// TwinCAT 3 PLC project Untitled1
// Title: RobustSolution
// Company: BATW
// Author: BATW
// ProjectVersion: 1.0.0.1
// ProgramVersion: 3.1.4026.24
// libraries:
//   Tc2_MC2, * (Beckhoff Automation GmbH)
//   Tc2_Standard, * (Beckhoff Automation GmbH)
//   Tc2_System, * (Beckhoff Automation GmbH)
//   Tc2_Utilities, * (Beckhoff Automation GmbH)
//   Tc3_JsonXml, * (Beckhoff Automation GmbH)
//   TcUnit, * (www.tcunit.org)
// project tree:
//   Configuration/DUTs/ E_AlarmOperator.TcDUT (not stored), E_ConfigDataType.TcDUT, E_ConfigValueError.TcDUT (not stored), E_LinkPhase.TcDUT (not stored), E_ModuleType.TcDUT, T_ModuleTypeName.TcDUT (not stored), E_VariableAccess.TcDUT, ST_ConfigRawValue.TcDUT (not stored), ST_ReferenceBindingFileConfig.TcDUT, ST_ConfigAlarmInfo.TcDUT (not stored), ST_ConfigVariableInfo.TcDUT (not stored), ST_RuntimeAlarmBinding.TcDUT (not stored), ST_RuntimeVariableBinding.TcDUT (not stored), ST_LinkVariableNode.TcDUT, ST_MappingFileConfig.TcDUT, ST_ModuleFileConfig.TcDUT, ST_ModuleRuntimeConfig.TcDUT, ST_SystemFileConfig.TcDUT, ST_VariableLink.TcDUT (not stored)
//   Configuration/POUs/ F_AlarmConditionMet.TcPOU, F_ConfigDataTypeSize.TcPOU, F_ConfigDataTypeToDescriptor.TcPOU (not stored), F_ConfigValueErrorMessage.TcPOU, FB_ConfigValueSnapshotReader.TcPOU, FB_ModuleTypeRegistry.TcPOU, FB_ReferenceManager.TcPOU, FB_ModuleReferenceBindingContext.TcPOU, FB_LinkVariableManager.TcPOU, FB_ModuleConfigurationManager.TcPOU, FB_ApplicationConfigRoot.TcPOU
//   Configuration/Interfaces/ I_AdsSymbolProvider.TcIO, I_ModuleReferenceBindings.TcIO, I_ModuleConfigurationAdapter.TcIO, I_VariableNodeReader.TcIO
//   DUTs/Contracts/Alarm/ E_Severity.TcDUT (not stored), ST_ExtAlarm.TcDUT (not stored)
//   DUTs/Contracts/Descriptor/ E_DescriptorType.TcDUT (not stored), ST_ExtDescriptor.TcDUT
//   DUTs/Contracts/System/ ST_SystemContext.TcDUT
//   DUTs/Infrastructure/EL Modules/ ST_EL1889Ex.TcDUT (not stored), ST_EL2809Ex.TcDUT (not stored), ST_EL3602Ex.TcDUT (not stored)
//   DUTs/Infrastructure/ ST_ReserveForGetSymbolNameByAddrress.TcDUT (not stored)
//   DUTs/Module/Alarm/ E_AlarmAckCommand.TcDUT (not stored), E_AlarmAckError.TcDUT (not stored), ST_AlarmAckRequest.TcDUT (not stored), ST_AlarmLifecycleState.TcDUT (not stored), ST_ModuleAlarmStatus.TcDUT (not stored)
//   DUTs/Module/Contract/ ST_ModuleCtrl.TcDUT (not stored), ST_ModuleDataStatus.TcDUT (not stored), ST_ModuleStatus.TcDUT (not stored), ST_ModuleVariableStatus.TcDUT, ST_Module_CtrlStatus_Base.TcDUT (not stored)
//   DUTs/Module/ServiceCoordination/ E_CompositeOwnershipState.TcDUT, E_ServiceCallSubmitResult.TcDUT, E_ServiceInternalCommandState.TcDUT (not stored), E_ServiceRegistrationError.TcDUT, ST_ServiceExecutionSnapshot.TcDUT, ST_ServiceRegistrationEntry.TcDUT
//   DUTs/Service/Composite/ E_CompositeServiceErrorCode.TcDUT
//   DUTs/Service/Contracts/ E_ServiceCompletionBehavior.TcDUT (not stored), ST_ServiceContext.TcDUT (not stored), ST_ServiceCtrl.TcDUT (not stored), ST_ServiceDataStatus.TcDUT, ST_ServiceExecuteSubStateRecord.TcDUT (not stored), ST_ServiceExecuteSubStateStatus.TcDUT, ST_ServiceStatus.TcDUT (not stored)
//   DUTs/Wafer Transfer/ E_OperationState.TcDUT (not stored), E_ReceiveState.TcDUT, E_TransferCapability.TcDUT, E_WaferHandlingType.TcDUT, ST_TransferHandshakeSignal.TcDUT, ST_MaterialContext.TcDUT, ST_MaterialInfo.TcDUT, ST_WaferTransferCtrl.TcDUT, ST_WaferTransferParam.TcDUT, ST_WaferTransferStatus.TcDUT, ST_WaferTransferResponse.TcDUT, ST_WaferTransferRequest.TcDUT
//   GVLs/ Param_Config.TcGVL
//   / PlcTask.TcTTO
//   POUs/00_BaseUnit/Base/ FB_BaseUnit.TcPOU (not stored), T_ResourceOwnerId.TcDUT (not stored)
//   POUs/00_BaseUnit/ FB_Axis_BaseUnit.TcPOU
//   POUs/00_BaseUnit/Interfaces/ I_Axis_BaseUnit.TcIO, I_BaseUnit.TcIO, I_ResourceLock.TcIO
//   POUs/10_Module/ FB_ModuleAlarmManager.TcPOU, FB_ModuleBase.TcPOU, FB_ServiceCoordinator.TcPOU, FB_ServiceCaller.TcPOU
//   POUs/20_Service/ FB_CompositeServiceBase.TcPOU (not stored), FB_ServiceBase.TcPOU (not stored)
//   POUs/ FB_UtcClock.TcPOU (not stored)
//   POUs/30_PackML_Base/DUTs/ E_PackMLCommand.TcDUT (not stored), E_PackMLErrorID.TcDUT (not stored), E_PackMLHookResult.TcDUT (not stored), E_PackMLMode.TcDUT (not stored), E_PackMLState.TcDUT (not stored), ST_PML_Base_In.TcDUT (not stored), ST_PML_Base_Out.TcDUT (not stored), T_PackMLMode.TcDUT
//   POUs/30_PackML_Base/ FB_PackMLBase.TcPOU, FB_PackMLModeSet.TcPOU (not stored)
//   POUs/30_PackML_Base/Utilities/ F_PackMLCommandToString.TcPOU (not stored), F_PackMLErrorIDToString.TcPOU (not stored), F_PackMLModeToString.TcPOU (not stored), F_PackMLStateToString.TcPOU (not stored)
// real-time tasks:
//   TASK PlcTask: cycle T#10ms, priority 20, ADS port 350

CONFIGURATION Untitled1
    RESOURCE PLC ON TwinCAT3
        TASK PlcTask(INTERVAL := T#10ms, PRIORITY := 20);
    END_RESOURCE
END_CONFIGURATION

// ---- Configuration/DUTs/E_ConfigDataType.TcDUT
{attribute 'qualified_only'}
{attribute 'strict'}
{attribute 'to_string'}
TYPE E_ConfigDataType :
(
	Unknown := 0,
	Boolean,
	Integer32,
	UnsignedInteger32,
	Float32,
	Float64,
	String80
);
END_TYPE

// ---- Configuration/DUTs/E_ModuleType.TcDUT
{attribute 'qualified_only'}
{attribute 'strict'}
{attribute 'to_string'}
TYPE E_ModuleType :
(
	Unknown := 0,
	// Chamber1 Module. The member name is the public config value.
	Chamber1 := 1
);
END_TYPE

// ---- Configuration/DUTs/E_VariableAccess.TcDUT
{attribute 'qualified_only'}
{attribute 'strict'}
TYPE E_VariableAccess :
(
	ReadOnly := 1,
	WriteOnly,
	ReadWrite
);
END_TYPE

// ---- Configuration/DUTs/ST_ReferenceBindingFileConfig.TcDUT
TYPE ST_ReferenceBindingFileConfig :
STRUCT
	Name : STRING(80);
	Source : STRING(255);
END_STRUCT
END_TYPE

// ---- Configuration/DUTs/ST_LinkVariableNode.TcDUT
TYPE ST_LinkVariableNode :
STRUCT
	Name : STRING(255);
	Address : PVOID;
	Size : UDINT;
	DataType : E_ConfigDataType;
	Access : E_VariableAccess;
END_STRUCT
END_TYPE

// ---- Configuration/DUTs/ST_MappingFileConfig.TcDUT
TYPE ST_MappingFileConfig :
STRUCT
	Source : STRING(255);
	Target : STRING(255);
	SourceDataType : E_ConfigDataType;
	TargetDataType : E_ConfigDataType;
	HasTransform : BOOL;
	Scale : LREAL;
	Offset : LREAL;
END_STRUCT
END_TYPE

// ---- Configuration/DUTs/ST_ModuleFileConfig.TcDUT
TYPE ST_ModuleFileConfig :
STRUCT
	Enabled : BOOL;
	Slot : UINT;
	Id : UDINT;
	ModuleType : T_ModuleTypeName;
	InputMappingCount : UINT;
	InputMappings : ARRAY[1..Param_Config.MaxModuleMappings] OF ST_MappingFileConfig;
	OutputMappingCount : UINT;
	OutputMappings : ARRAY[1..Param_Config.MaxModuleMappings] OF ST_MappingFileConfig;
	ReferenceCount : UINT;
	References : ARRAY[1..Param_Config.MaxModuleReferences] OF ST_ReferenceBindingFileConfig;
	VariableCount : UINT;
	VariableList : ARRAY[1..Param_Config.MaxModuleVariable] OF ST_ConfigVariableInfo;
	AlarmCount : UINT;
	AlarmList : ARRAY[1..Param_Config.MaxConfiguredAlarmsPerModule] OF ST_ConfigAlarmInfo;
END_STRUCT
END_TYPE

// ---- Configuration/DUTs/ST_ModuleRuntimeConfig.TcDUT
TYPE ST_ModuleRuntimeConfig :
STRUCT
	Enabled : BOOL;
	Valid : BOOL;
	ModuleId : UDINT;
	ModuleType : T_ModuleTypeName;
	Revision : UDINT;
	VariableCount : UINT;
	VariableBindings : ARRAY[1..Param_Config.MaxModuleVariable] OF ST_RuntimeVariableBinding;
	AlarmCount : UINT;
	AlarmBindings : ARRAY[1..Param_Config.MaxConfiguredAlarmsPerModule] OF ST_RuntimeAlarmBinding;
END_STRUCT
END_TYPE

// ---- Configuration/DUTs/ST_SystemFileConfig.TcDUT
TYPE ST_SystemFileConfig :
STRUCT
	SchemaVersion : UDINT;
	ModuleCount : UINT;
	Modules : ARRAY[1..Param_Config.MaxTotalConfiguredModules] OF ST_ModuleFileConfig;
END_STRUCT
END_TYPE

// ---- DUTs/Contracts/Descriptor/ST_ExtDescriptor.TcDUT
TYPE ST_ExtDescriptor :
STRUCT
	Id : UDINT;
	Name : STRING(30);
	DataType : E_DescriptorType;
	Unit : STRING(10);
	Value : STRING(80);
END_STRUCT
END_TYPE

// ---- DUTs/Contracts/System/ST_SystemContext.TcDUT
TYPE ST_SystemContext :
STRUCT
	// UTC timestamp formatted as YYYYMMDDHHMMSSUUU.
	UtcDateTime : STRING(20);
	// Maximum time that a Module may observe an unchanged HeartbeatIndex.
	ModuleHeartbeatTimeout : TIME;
END_STRUCT
END_TYPE

// ---- DUTs/Module/Contract/ST_ModuleVariableStatus.TcDUT
TYPE ST_ModuleVariableStatus :
STRUCT
	PublishedCount : UINT;
	Overflow : BOOL;
	DuplicateId : UDINT;
END_STRUCT
END_TYPE

// ---- DUTs/Module/ServiceCoordination/E_CompositeOwnershipState.TcDUT
{attribute 'qualified_only'}
{attribute 'strict'}
{attribute 'to_string'}
TYPE E_CompositeOwnershipState :
(
	None := 0,
	Pending := 1,
	Owned := 2,
	RejectedConflict := 3,
	RejectedDependencyNotIdle := 4,
	RejectedUnsupportedCompletionBehavior := 5,
	Cancelled := 6
) UDINT;
END_TYPE

// ---- DUTs/Module/ServiceCoordination/E_ServiceCallSubmitResult.TcDUT
{attribute 'qualified_only'}
{attribute 'strict'}
{attribute 'to_string'}
TYPE E_ServiceCallSubmitResult :
(
	Queued := 0,
	CallerNotConfigured := 1,
	CoordinatorNotReady := 2,
	UnknownService := 3,
	DependencyNotDeclared := 4,
	NotOwner := 5,
	Busy := 6,
	InvalidCommand := 7,
	ParameterSizeMismatch := 8,
	ParameterTypeResolutionFailed := 9,
	ParameterTypeMismatch := 10
) UDINT;
END_TYPE

// ---- DUTs/Module/ServiceCoordination/E_ServiceRegistrationError.TcDUT
{attribute 'qualified_only'}
{attribute 'strict'}
{attribute 'to_string'}
TYPE E_ServiceRegistrationError :
(
	None := 0,
	RegistrationAlreadyStarted := 1,
	RegistryAlreadySealed := 2,
	EmptyRegistry := 3,
	CapacityExceeded := 4,
	InvalidServiceId := 5,
	DuplicateServiceId := 6,
	InvalidStorage := 7,
	ParameterSizeMismatch := 8,
	ParameterTypeMismatch := 9,
	ParameterTypeResolutionFailed := 10,
	InvalidCompositeService := 11,
	DuplicateCompositeDefinition := 12,
	EmptyCompositeDependencyList := 13,
	CompositeDependencyCapacityExceeded := 14,
	InvalidCompositeDependencyId := 15,
	UnknownCompositeDependency := 16,
	SelfDependency := 17,
	DuplicateCompositeDependency := 18,
	CompositeDependencyNotAllowed := 19,
	NestedCompositeNotSupported := 20
) UDINT;
END_TYPE

// ---- DUTs/Module/ServiceCoordination/ST_ServiceExecutionSnapshot.TcDUT
TYPE ST_ServiceExecutionSnapshot :
STRUCT
	Valid : BOOL;
	ServiceId : UDINT;
	ResponseId : UDINT;
	PackMLOut : ST_PML_Base_Out;
	ExecuteSubState : UDINT;
	CompletionBehavior : E_ServiceCompletionBehavior;
END_STRUCT
END_TYPE

// ---- DUTs/Module/ServiceCoordination/ST_ServiceRegistrationEntry.TcDUT
TYPE ST_ServiceRegistrationEntry :
STRUCT
	InUse : BOOL;
	ServiceId : UDINT;

	UpperCtrlAddress : PVOID;
	EffectiveCtrlAddress : PVOID;

	UpperParamAddress : PVOID;
	EffectiveParamAddress : PVOID;
	ParameterSize : UDINT;
	ParameterTypeName : STRING(255);

	StatusAddress : PVOID;
	AllowCompositeCall : BOOL;
	IsComposite : BOOL;
	CompositeOwnerServiceId : UDINT;

	CompositeDependenciesAddress : PVOID;
	CompositeDependencyCount : UINT;
	OwnershipState : E_CompositeOwnershipState;

	InternalRequestId : UDINT;
	InternalCommand : E_PackMLCommand;
	InternalCommandState : E_ServiceInternalCommandState;
	InternalRequestMustGoLow : BOOL;

	ObservedSnapshot : ST_ServiceExecutionSnapshot;

	UpperCommandWasHigh : BOOL;
	UpperModeWasHigh : BOOL;
	UpperCommandBlockedUntilFalse : BOOL;
	UpperModeBlockedUntilFalse : BOOL;
END_STRUCT
END_TYPE

// ---- DUTs/Service/Composite/E_CompositeServiceErrorCode.TcDUT
{attribute 'qualified_only'}
{attribute 'strict'}
{attribute 'to_string'}
TYPE E_CompositeServiceErrorCode :
(
	None := 0,
	NotConfigured := 1,
	OwnershipConflict := 2,
	DependencyNotIdle := 3,
	UnsupportedCompletionBehavior := 4,
	InternalCallSubmitFailed := 5,
	InternalCommandRejected := 6,
	ChildStoppedUnexpectedly := 7,
	ChildAbortedUnexpectedly := 8,
	SequenceFailed := 9,
	InvalidSequenceState := 10
) UDINT;
END_TYPE

// ---- DUTs/Service/Contracts/ST_ServiceDataStatus.TcDUT
TYPE ST_ServiceDataStatus :
STRUCT
	Count : UINT;
	Overflow : BOOL;
	DataList : ARRAY[1..Param_Config.MaxServiceData] OF ST_ExtDescriptor;
END_STRUCT
END_TYPE

// ---- DUTs/Service/Contracts/ST_ServiceExecuteSubStateStatus.TcDUT
TYPE ST_ServiceExecuteSubStateStatus :
STRUCT
	// Zero whenever the Service is not executing or exposes no substate.
	CurrentState : UDINT;
	RecordCount : UINT;
	// The first records are preserved when capacity is exhausted.
	Overflow : BOOL;
	Records : ARRAY[1..Param_Config.MaxExecuteSubStateRecords] OF ST_ServiceExecuteSubStateRecord;
END_STRUCT
END_TYPE

// ---- DUTs/Wafer Transfer/E_ReceiveState.TcDUT
{attribute 'qualified_only'}
{attribute 'strict'}
{attribute 'to_string'}
TYPE E_ReceiveState :
(
	None := 0,
	Candidate,
	Bound,
	Commited
);
END_TYPE

// ---- DUTs/Wafer Transfer/E_TransferCapability.TcDUT
{attribute 'qualified_only'}
{attribute 'strict'}
{attribute 'to_string'}
TYPE E_TransferCapability :
(
	Unknown := 0,
	SendOnly,
	ReveiveOnly,
	Bidirectional
);
END_TYPE

// ---- DUTs/Wafer Transfer/E_WaferHandlingType.TcDUT
{attribute 'qualified_only'}
{attribute 'strict'}
{attribute 'to_string'}
TYPE E_WaferHandlingType :
(
	Unknown := 0,
	Passive,
	Active
);
END_TYPE

// ---- DUTs/Wafer Transfer/ST_TransferHandshakeSignal.TcDUT
TYPE ST_TransferHandshakeSignal :
STRUCT
	Accept : BOOL;
	Ready : BOOL;
	ReceiveRequest : BOOL;
	SendRequest : BOOL;
	SendComplete : BOOL;
	ReceiveComplete : BOOL;
END_STRUCT
END_TYPE

// ---- DUTs/Wafer Transfer/ST_MaterialContext.TcDUT
TYPE ST_MaterialContext :
STRUCT
	Id : UDINT;
	// Add other information of wafer...
END_STRUCT
END_TYPE

// ---- DUTs/Wafer Transfer/ST_MaterialInfo.TcDUT
TYPE ST_MaterialInfo :
STRUCT
	MaterialPresence : BOOL;	// Could be sensor signal
	OwnerShip : BOOL;			// Pure software logic
	ReceiveState : E_ReceiveState;
	OperationState : E_OperationState;
	MaterialContext : ST_MaterialContext;
END_STRUCT
END_TYPE

// ---- DUTs/Wafer Transfer/ST_WaferTransferCtrl.TcDUT
TYPE ST_WaferTransferCtrl :
STRUCT
	Ctrl : ST_ServiceCtrl;
	Param : ST_WaferTransferParam;
	Signal : ST_TransferHandshakeSignal;
END_STRUCT
END_TYPE

// ---- DUTs/Wafer Transfer/ST_WaferTransferParam.TcDUT
TYPE ST_WaferTransferParam :
STRUCT
	MaterialContext : ST_MaterialContext;
	Signal : ST_TransferHandshakeSignal;
END_STRUCT
END_TYPE

// ---- DUTs/Wafer Transfer/ST_WaferTransferStatus.TcDUT
TYPE ST_WaferTransferStatus :
STRUCT
	Status : ST_ServiceStatus;
	Signal : ST_TransferHandshakeSignal;
END_STRUCT
END_TYPE

// ---- DUTs/Wafer Transfer/ST_WaferTransferResponse.TcDUT
TYPE ST_WaferTransferResponse :
STRUCT
	// Managed by module
	// Non-zero and unique within one Module; array index is storage only.
	EndpointId : UDINT;
	SendServiceId : UDINT;
	ReceiveServiceId : UDINT;
	WaferHandlingType : E_WaferHandlingType;
	Capability : E_TransferCapability;

	// Managed by module
	// Passive only (both can be TRUE in multi-station chamber)
	SendReady : BOOL;
	ReceiveReady : BOOL;
	
	// Managed by service
	Send : ST_WaferTransferStatus;
	Receive : ST_WaferTransferStatus;
	
	MaterialInfo : ST_MaterialInfo;
END_STRUCT
END_TYPE

// ---- DUTs/Wafer Transfer/ST_WaferTransferRequest.TcDUT
TYPE ST_WaferTransferRequest :
STRUCT
	Send : ST_WaferTransferCtrl;
	Receive : ST_WaferTransferCtrl;
END_STRUCT
END_TYPE

// ---- POUs/30_PackML_Base/DUTs/T_PackMLMode.TcDUT
TYPE T_PackMLMode : UINT;
END_TYPE

// ---- GVLs/Param_Config.TcGVL
{attribute 'qualified_only'}
VAR_GLOBAL CONSTANT
	MaxModuleVariable : UINT := 100;	// Num of SVID
	MaxConfiguredAlarmsPerModule : UINT := 30;	// Num of configured ALIDs.
	MaxHookAlarmsPerModule : UINT := 30;		// Reserved capacity for Module Hook alarms.
	MaxServiceAlarmsPerModule : UINT := 40;		// Reserved capacity for aggregated Service errors.
	MaxPublishedModuleAlarms : UINT := MaxConfiguredAlarmsPerModule + MaxHookAlarmsPerModule + MaxServiceAlarmsPerModule;
	MaxModuleAlarm : UINT := MaxPublishedModuleAlarms;	// Compatibility alias for existing consumers.
	MaxServiceError : UINT := 10;		// Num of Service Error per round
	MaxServiceData : UINT := 30;		// Num of persistent Data descriptors per Service
	MaxServicesPerModule : UINT := 100;	// Maximum number of Services registered by one Module.
	MaxCompositeDependencies : UINT := 10;	// Maximum number of child Services declared by one Composite Service.
	MaxModuleData : UINT := 50;			// Num of DVID
	MaxTransferEndpoint : UINT := 2;	// Num of wafer transfer port
	MaxProcessStation : UINT := 4;		// Num of wafer process station
	ModuleHeartbeat_Timeout : TIME := T#10S;

	// Runtime configuration limits. They also bound PLC memory and local snapshot work.
	MaxModuleTypes : UINT := 8;

	// Module type capacities bound type-specific runtime arrays.
	MaxModulePerType : UINT := 6;

	// Total config capacity is the compile-time sum of every supported Module type capacity.
	MaxTotalConfiguredModules : UINT := MaxModulePerType * MaxModuleTypes;

	// Variable mapping
	MaxModuleMappings : UINT := 256;
	MaxConfigVariableNodes : UINT := 512;

	// Reference binding
	MaxModuleReferences : UINT := 50;
	MaxConfigReferenceNodes : UINT := 100;

	// Registered-node snapshots used by configured VariableList and AlarmList.
	MaxConfiguredValueSources : UINT := MaxModuleVariable + MaxConfiguredAlarmsPerModule;
	MaxConfigValueSize : UINT := 81; // STRING(80), including the terminating zero.

	// System config
	ConfigSchemaVersion : UDINT := 4;
	ModuleConfigFilePath : STRING(255) := 'C:\ProgramData\RobustSolution\module-config.json';
END_VAR

// ---- Configuration/Interfaces/I_AdsSymbolProvider.TcIO
INTERFACE I_AdsSymbolProvider EXTENDS __SYSTEM.IQueryInterface

METHOD M_GetAdsSymbolMetadata : BOOL
VAR_OUTPUT
	Address : PVOID;
	Size : UDINT;
END_VAR
END_METHOD

END_INTERFACE

// ---- Configuration/Interfaces/I_ModuleReferenceBindings.TcIO
INTERFACE I_ModuleReferenceBindings EXTENDS __SYSTEM.IQueryInterface

METHOD M_TakeOptional : I_BaseUnit
VAR_INPUT
	Port : ANY;
END_VAR
VAR_OUTPUT
	PortName : STRING(80);
	Present : BOOL;
	ErrorMessage : STRING(255);
END_VAR
END_METHOD

METHOD M_TakeRequired : I_BaseUnit
VAR_INPUT
	Port : ANY;
END_VAR
VAR_OUTPUT
	PortName : STRING(80);
	ErrorMessage : STRING(255);
END_VAR
END_METHOD

METHOD M_SetModuleScope : BOOL
VAR_INPUT
	ModuleSymbol : STRING(255);
END_VAR
VAR_OUTPUT
	ErrorMessage : STRING(255);
END_VAR
END_METHOD

END_INTERFACE

// ---- Configuration/Interfaces/I_ModuleConfigurationAdapter.TcIO
INTERFACE I_ModuleConfigurationAdapter EXTENDS __SYSTEM.IQueryInterface

METHOD M_ApplyRuntimeConfig : BOOL
VAR_INPUT
	Slot : UINT;
END_VAR
VAR_IN_OUT CONSTANT
	RuntimeConfig : ST_ModuleRuntimeConfig;
END_VAR
VAR_OUTPUT
	ErrorMessage : STRING(255);
END_VAR
END_METHOD

METHOD M_ClearAllSlots : BOOL
VAR_OUTPUT
	ErrorMessage : STRING(255);
END_VAR
END_METHOD

METHOD M_IsSlotSupported : BOOL
VAR_INPUT
	Slot : UINT;
END_VAR
END_METHOD

METHOD M_PrepareInstance : BOOL
VAR_INPUT
	Slot : UINT;
	ReferenceBindings : I_ModuleReferenceBindings;
END_VAR
VAR_IN_OUT
	ModuleConfig : ST_ModuleFileConfig;
	LinkVariableManager : FB_LinkVariableManager;
END_VAR
VAR_OUTPUT
	ModuleSymbol : STRING(255);
	ErrorMessage : STRING(255);
END_VAR
END_METHOD

END_INTERFACE

// ---- Configuration/Interfaces/I_VariableNodeReader.TcIO
INTERFACE I_VariableNodeReader EXTENDS __SYSTEM.IQueryInterface

METHOD M_ReadNode : BOOL
VAR_INPUT
	NodeHandle : UINT;
	ExpectedDataType : E_ConfigDataType;
END_VAR
VAR_IN_OUT
	Value : ST_ConfigRawValue;
END_VAR
VAR_OUTPUT
	ErrorCode : E_ConfigValueError;
END_VAR
END_METHOD

END_INTERFACE

// ---- POUs/00_BaseUnit/Interfaces/I_Axis_BaseUnit.TcIO
INTERFACE I_Axis_BaseUnit EXTENDS I_ResourceLock

PROPERTY AxisActualPosition : LREAL
GET
END_GET
END_PROPERTY

PROPERTY AxisActualVelocity : LREAL
GET
END_GET
END_PROPERTY

PROPERTY AxisHasJob : BOOL
GET
END_GET
END_PROPERTY

PROPERTY AxisIsDisabled : BOOL
GET
END_GET
END_PROPERTY

METHOD M_CyclicUpdate
VAR_INPUT
END_VAR
END_METHOD

METHOD M_Halt : BOOL
VAR_INPUT
	OwnerId : T_ResourceOwnerId;
	Execute : BOOL;
	Deceleration : LREAL;
END_VAR
VAR_OUTPUT
	Done : BOOL;
	Error : BOOL;
END_VAR
END_METHOD

METHOD M_Jog : BOOL
VAR_INPUT
	OwnerId : T_ResourceOwnerId;
	JogForward : BOOL;
	JogBackwards : BOOL;
	Mode : E_JogMode;
	Position : LREAL;
	Velocity : LREAL;
	Acceleration : LREAL;
	Deceleration : LREAL;
END_VAR
VAR_OUTPUT
	Done : BOOL;
	Error : BOOL;
	ErrorId : UDINT;
END_VAR
END_METHOD

METHOD M_MoveAbs : BOOL
VAR_INPUT
	OwnerId : T_ResourceOwnerId;
	Execute : BOOL;
	Position : LREAL;
	Velocity : LREAL;
	Acceleration : LREAL;
	Deceleration : LREAL;
END_VAR
VAR_OUTPUT
	Done : BOOL;
	Error : BOOL;
	ErrorId : UDINT;
END_VAR
END_METHOD

METHOD M_MoveVel : BOOL
VAR_INPUT
	OwnerId : T_ResourceOwnerId;
	Execute : BOOL;
	Direction : MC_Direction;
	Velocity : LREAL;
	Acceleration : LREAL;
	Deceleration : LREAL;
END_VAR
VAR_OUTPUT
	InVelocity : BOOL;
	Error : BOOL;
END_VAR
END_METHOD

METHOD M_Reset : BOOL
VAR_INPUT
	OwnerId : T_ResourceOwnerId;
	Execute : BOOL;
END_VAR
VAR_OUTPUT
	Done : BOOL;
	Error : BOOL;
	ErrorId : UDINT;
END_VAR
END_METHOD

METHOD M_Stop : BOOL
VAR_INPUT
	OwnerId : T_ResourceOwnerId;
	Execute : BOOL;
	Deceleration : LREAL;
END_VAR
VAR_OUTPUT
	Done : BOOL;
	Error : BOOL;
	ErrorId : UDINT;
END_VAR
END_METHOD

END_INTERFACE

// ---- POUs/00_BaseUnit/Interfaces/I_BaseUnit.TcIO
INTERFACE I_BaseUnit EXTENDS __SYSTEM.IQueryInterface

END_INTERFACE

// ---- POUs/00_BaseUnit/Interfaces/I_ResourceLock.TcIO
INTERFACE I_ResourceLock

METHOD M_AcquireResource : BOOL
VAR_INPUT
	OwnerId : T_ResourceOwnerId;
END_VAR
END_METHOD

METHOD M_IsResourceOwner : BOOL
VAR_INPUT
	OwnerId : T_ResourceOwnerId;
END_VAR
END_METHOD

METHOD M_ReleaseResource : BOOL
VAR_INPUT
	OwnerId : T_ResourceOwnerId;
END_VAR
END_METHOD

END_INTERFACE

// ---- Configuration/POUs/F_AlarmConditionMet.TcPOU
FUNCTION F_AlarmConditionMet : BOOL
VAR_INPUT
	Value : LREAL;
	Operator : E_AlarmOperator;
	Threshold : LREAL;
	Tolerance : LREAL;
END_VAR
VAR
	fTolerance : LREAL;
END_VAR

fTolerance := ABS(Tolerance);

CASE Operator OF
	E_AlarmOperator.GreaterThan:
		F_AlarmConditionMet := Value > Threshold;
	E_AlarmOperator.LessThan:
		F_AlarmConditionMet := Value < Threshold;
	E_AlarmOperator.Equal:
		F_AlarmConditionMet := ABS(Value - Threshold) <= fTolerance;
	E_AlarmOperator.GreaterOrEqual:
		F_AlarmConditionMet := Value >= Threshold;
	E_AlarmOperator.LessOrEqual:
		F_AlarmConditionMet := Value <= Threshold;
ELSE
	F_AlarmConditionMet := FALSE;
END_CASE

END_FUNCTION

// ---- Configuration/POUs/F_ConfigDataTypeSize.TcPOU
FUNCTION F_ConfigDataTypeSize : UDINT
VAR_INPUT
	DataType : E_ConfigDataType;
END_VAR

CASE DataType OF
	E_ConfigDataType.Boolean:
		F_ConfigDataTypeSize := SIZEOF(BOOL);
	E_ConfigDataType.Integer32:
		F_ConfigDataTypeSize := SIZEOF(DINT);
	E_ConfigDataType.UnsignedInteger32:
		F_ConfigDataTypeSize := SIZEOF(UDINT);
	E_ConfigDataType.Float32:
		F_ConfigDataTypeSize := SIZEOF(REAL);
	E_ConfigDataType.Float64:
		F_ConfigDataTypeSize := SIZEOF(LREAL);
	E_ConfigDataType.String80:
		F_ConfigDataTypeSize := 81;
ELSE
	F_ConfigDataTypeSize := 0;
END_CASE

END_FUNCTION

// ---- Configuration/POUs/F_ConfigValueErrorMessage.TcPOU
FUNCTION F_ConfigValueErrorMessage : STRING(160)
VAR_INPUT
	ErrorCode : E_ConfigValueError;
END_VAR

CASE ErrorCode OF
	E_ConfigValueError.None:
		F_ConfigValueErrorMessage := '';
	E_ConfigValueError.ReaderUnavailable:
		F_ConfigValueErrorMessage := 'Variable node reader is not available.';
	E_ConfigValueError.SourceCapacityExceeded:
		F_ConfigValueErrorMessage := 'Configured value source count exceeds snapshot capacity.';
	E_ConfigValueError.InvalidNodeHandle:
		F_ConfigValueErrorMessage := 'Configured value node handle is invalid.';
	E_ConfigValueError.NodeReadNotAllowed:
		F_ConfigValueErrorMessage := 'Configured value node is write-only.';
	E_ConfigValueError.InvalidNodeAddress:
		F_ConfigValueErrorMessage := 'Configured value node address is invalid.';
	E_ConfigValueError.NodeDataTypeMismatch:
		F_ConfigValueErrorMessage := 'Configured value type does not match the registered node.';
	E_ConfigValueError.InvalidNodeSize:
		F_ConfigValueErrorMessage := 'Configured value node size is invalid or exceeds the snapshot buffer.';
ELSE
	F_ConfigValueErrorMessage := 'Unknown configured value read error.';
END_CASE

END_FUNCTION

// ---- Configuration/POUs/FB_ConfigValueSnapshotReader.TcPOU
FUNCTION_BLOCK FB_ConfigValueSnapshotReader
VAR_INPUT
	RuntimeConfig : REFERENCE TO ST_ModuleRuntimeConfig;
	VariableNodeReader : I_VariableNodeReader;
END_VAR
VAR_OUTPUT
	Ready : BOOL;
	Error : BOOL;
	ErrorCode : E_ConfigValueError;
	ErrorMessage : STRING(255);
	ErrorSource : STRING(255);
END_VAR
VAR
	_SourceCount : UINT;
	_SourceTypes : ARRAY[1..Param_Config.MaxConfiguredValueSources] OF E_ConfigDataType;
	_Values : ARRAY[1..Param_Config.MaxConfiguredValueSources] OF ST_ConfigRawValue;
	_ValueValid : ARRAY[1..Param_Config.MaxConfiguredValueSources] OF BOOL;

END_VAR
VAR_TEMP
	_nIndex : UINT;
	_nSource : UINT;
	_eReadError : E_ConfigValueError;
END_VAR

Ready := FALSE;
Error := FALSE;
ErrorCode := E_ConfigValueError.None;
ErrorMessage := '';
ErrorSource := '';
_SourceCount := 0;

IF NOT __ISVALIDREF(RuntimeConfig) THEN
	RETURN;
END_IF
IF NOT RuntimeConfig.Enabled OR NOT RuntimeConfig.Valid THEN
	RETURN;
END_IF
IF VariableNodeReader = 0 THEN
	M_SetFirstError(
		ErrorCodeValue := E_ConfigValueError.ReaderUnavailable,
		SourceName := '');
	RETURN;
END_IF

_SourceCount := RuntimeConfig.VariableCount + RuntimeConfig.AlarmCount;
IF _SourceCount > Param_Config.MaxConfiguredValueSources THEN
	M_SetFirstError(
		ErrorCodeValue := E_ConfigValueError.SourceCapacityExceeded,
		SourceName := '');
	RETURN;
END_IF

MEMSET(ADR(_SourceTypes), 0, SIZEOF(_SourceTypes));
MEMSET(ADR(_ValueValid), 0, SIZEOF(_ValueValid));

FOR _nIndex := 1 TO RuntimeConfig.VariableCount DO
	_nSource := _nIndex;
	_SourceTypes[_nSource] := RuntimeConfig.VariableBindings[_nIndex].Definition.DataType;
	_ValueValid[_nSource] := VariableNodeReader.M_ReadNode(
		NodeHandle := RuntimeConfig.VariableBindings[_nIndex].NodeHandle,
		ExpectedDataType := _SourceTypes[_nSource],
		Value := _Values[_nSource],
		ErrorCode => _eReadError);
	IF NOT _ValueValid[_nSource] AND NOT Error THEN
		M_SetFirstError(
			ErrorCodeValue := _eReadError,
			SourceName := RuntimeConfig.VariableBindings[_nIndex].Definition.Source);
	END_IF
END_FOR

FOR _nIndex := 1 TO RuntimeConfig.AlarmCount DO
	_nSource := RuntimeConfig.VariableCount + _nIndex;
	_SourceTypes[_nSource] := RuntimeConfig.AlarmBindings[_nIndex].Definition.DataType;
	_ValueValid[_nSource] := VariableNodeReader.M_ReadNode(
		NodeHandle := RuntimeConfig.AlarmBindings[_nIndex].NodeHandle,
		ExpectedDataType := _SourceTypes[_nSource],
		Value := _Values[_nSource],
		ErrorCode => _eReadError);
	IF NOT _ValueValid[_nSource] AND NOT Error THEN
		M_SetFirstError(
			ErrorCodeValue := _eReadError,
			SourceName := RuntimeConfig.AlarmBindings[_nIndex].Definition.Source);
	END_IF
END_FOR

Ready := NOT Error;

METHOD PRIVATE M_SetFirstError
VAR_INPUT
	ErrorCodeValue : E_ConfigValueError;
	SourceName : STRING(255);
END_VAR
IF Error THEN
	RETURN;
END_IF

Error := TRUE;
ErrorCode := ErrorCodeValue;
ErrorMessage := F_ConfigValueErrorMessage(ErrorCode := ErrorCodeValue);
ErrorSource := SourceName;
END_METHOD

METHOD PUBLIC M_GetLReal : LREAL
VAR_INPUT
	SourceIndex : UINT;
END_VAR
VAR_OUTPUT
	Valid : BOOL;
END_VAR
VAR
	pBool : POINTER TO BOOL;
	pDInt : POINTER TO DINT;
	pUDInt : POINTER TO UDINT;
	pReal : POINTER TO REAL;
	pLReal : POINTER TO LREAL;
END_VAR
Valid := FALSE;
M_GetLReal := 0.0;
IF NOT Ready OR (SourceIndex < 1) OR (SourceIndex > _SourceCount)
	OR NOT _ValueValid[SourceIndex] THEN
	RETURN;
END_IF

CASE _SourceTypes[SourceIndex] OF
	E_ConfigDataType.Boolean:
		pBool := ADR(_Values[SourceIndex].Data);
		IF pBool^ THEN M_GetLReal := 1.0; END_IF
	E_ConfigDataType.Integer32:
		pDInt := ADR(_Values[SourceIndex].Data);
		M_GetLReal := DINT_TO_LREAL(pDInt^);
	E_ConfigDataType.UnsignedInteger32:
		pUDInt := ADR(_Values[SourceIndex].Data);
		M_GetLReal := UDINT_TO_LREAL(pUDInt^);
	E_ConfigDataType.Float32:
		pReal := ADR(_Values[SourceIndex].Data);
		M_GetLReal := REAL_TO_LREAL(pReal^);
	E_ConfigDataType.Float64:
		pLReal := ADR(_Values[SourceIndex].Data);
		M_GetLReal := pLReal^;
ELSE
	RETURN;
END_CASE
Valid := TRUE;
END_METHOD

METHOD PUBLIC M_GetValueString : STRING(80)
VAR_INPUT
	SourceIndex : UINT;
END_VAR
VAR_OUTPUT
	Valid : BOOL;
END_VAR
VAR
	pBool : POINTER TO BOOL;
	pDInt : POINTER TO DINT;
	pUDInt : POINTER TO UDINT;
	pReal : POINTER TO REAL;
	pLReal : POINTER TO LREAL;
	sValue : STRING(80);
END_VAR
Valid := FALSE;
M_GetValueString := '';
IF NOT Ready OR (SourceIndex < 1) OR (SourceIndex > _SourceCount)
	OR NOT _ValueValid[SourceIndex] THEN
	RETURN;
END_IF

CASE _SourceTypes[SourceIndex] OF
	E_ConfigDataType.Boolean:
		pBool := ADR(_Values[SourceIndex].Data);
		sValue := BOOL_TO_STRING(pBool^);
	E_ConfigDataType.Integer32:
		pDInt := ADR(_Values[SourceIndex].Data);
		sValue := DINT_TO_STRING(pDInt^);
	E_ConfigDataType.UnsignedInteger32:
		pUDInt := ADR(_Values[SourceIndex].Data);
		sValue := UDINT_TO_STRING(pUDInt^);
	E_ConfigDataType.Float32:
		pReal := ADR(_Values[SourceIndex].Data);
		sValue := REAL_TO_STRING(pReal^);
	E_ConfigDataType.Float64:
		pLReal := ADR(_Values[SourceIndex].Data);
		sValue := LREAL_TO_STRING(pLReal^);
	E_ConfigDataType.String80:
		MEMCPY(ADR(sValue), ADR(_Values[SourceIndex].Data), SIZEOF(sValue));
ELSE
	RETURN;
END_CASE
M_GetValueString := sValue;
Valid := TRUE;
END_METHOD

END_FUNCTION_BLOCK

// ---- Configuration/POUs/FB_ModuleTypeRegistry.TcPOU
FUNCTION_BLOCK FB_ModuleTypeRegistry
VAR_OUTPUT
	Error : BOOL;
	ErrorMessage : STRING(255);
END_VAR
VAR
	_ModuleTypes : ARRAY[1..Param_Config.MaxModuleTypes] OF T_ModuleTypeName;
	_Adapters : ARRAY[1..Param_Config.MaxModuleTypes] OF I_ModuleConfigurationAdapter;
	_Count : UINT;
END_VAR

METHOD PUBLIC M_ClearAll : BOOL
VAR
	nAdapter : UINT;
	sAdapterError : STRING(255);
END_VAR
M_ClearAll := FALSE;
Error := FALSE;
ErrorMessage := '';
FOR nAdapter := 1 TO _Count DO
	IF NOT _Adapters[nAdapter].M_ClearAllSlots(
		ErrorMessage => sAdapterError) THEN
		Error := TRUE;
		ErrorMessage := sAdapterError;
		RETURN;
	END_IF
END_FOR
M_ClearAll := TRUE;
END_METHOD

METHOD PUBLIC M_Register : BOOL
VAR_INPUT
	ModuleTypeName : T_ModuleTypeName;
	Adapter : I_ModuleConfigurationAdapter;
END_VAR
VAR
	nIndex : UINT;
END_VAR
M_Register := FALSE;
Error := FALSE;
ErrorMessage := '';
IF (ModuleTypeName = '') OR (Adapter = 0) THEN
	Error := TRUE;
	ErrorMessage := 'A Module Type name and adapter are required.';
	RETURN;
END_IF

FOR nIndex := 1 TO _Count DO
	IF _ModuleTypes[nIndex] = ModuleTypeName THEN
		_Adapters[nIndex] := Adapter;
		M_Register := TRUE;
		RETURN;
	END_IF
END_FOR

nIndex := _Count + 1;
IF nIndex > Param_Config.MaxModuleTypes THEN
	Error := TRUE;
	ErrorMessage := 'Module type registry is full.';
	RETURN;
END_IF
_ModuleTypes[nIndex] := ModuleTypeName;
_Adapters[nIndex] := Adapter;
_Count := nIndex;
M_Register := TRUE;
END_METHOD

METHOD PUBLIC M_Resolve : I_ModuleConfigurationAdapter
VAR_INPUT
	ModuleTypeName : T_ModuleTypeName;
END_VAR
VAR
	nIndex : UINT;
END_VAR
M_Resolve := 0;
Error := FALSE;
ErrorMessage := '';
FOR nIndex := 1 TO _Count DO
	IF ModuleTypeName = _ModuleTypes[nIndex] THEN
		M_Resolve := _Adapters[nIndex];
		RETURN;
	END_IF
END_FOR
Error := TRUE;
ErrorMessage := 'Module type was not registered.';
END_METHOD

END_FUNCTION_BLOCK

// ---- Configuration/POUs/FB_ReferenceManager.TcPOU
FUNCTION_BLOCK FB_ReferenceManager
VAR_OUTPUT
	Error : BOOL;
	ErrorMessage : STRING(255);
END_VAR
VAR
	_JsonDataType : FB_JsonReadWriteDataType;
	_Names : ARRAY[1..Param_Config.MaxConfigReferenceNodes] OF STRING(255);
	_BaseUnits : ARRAY[1..Param_Config.MaxConfigReferenceNodes] OF I_BaseUnit;
	_Count : UINT;
END_VAR

METHOD PUBLIC M_RegisterReference : BOOL
VAR_INPUT
	BaseUnit : I_BaseUnit;
END_VAR
VAR
	nIndex : UINT;
	sName : STRING(255);
	pData : PVOID;
	nData : UDINT;
	SymbolProvider : I_AdsSymbolProvider;
	hrErrorCode : HRESULT;
END_VAR
M_RegisterReference := FALSE;
Error := FALSE;
ErrorMessage := '';
IF BaseUnit = 0 THEN
	Error := TRUE;
	ErrorMessage := 'Cannot register an unbound BaseUnit interface.';
	RETURN;
END_IF

SymbolProvider := 0;
IF NOT __QUERYINTERFACE(BaseUnit, SymbolProvider) THEN
	Error := TRUE;
	ErrorMessage := 'BaseUnit does not provide ADS symbol metadata.';
	RETURN;
END_IF

// Get address & size
IF NOT SymbolProvider.M_GetAdsSymbolMetadata(
	Address => pData,
	Size => nData) THEN
	Error := TRUE;
	ErrorMessage := 'BaseUnit ADS symbol metadata is invalid.';
	RETURN;
END_IF

// Get symbol name by address&size
sName := _JsonDataType.GetSymbolNameByAddress(
	nData := nData,
	pData := pData,
	hrErrorCode => hrErrorCode);
IF (hrErrorCode <> 0) OR (sName = '') THEN
	Error := TRUE;
	ErrorMessage := 'Cannot resolve the BaseUnit ADS symbol name.';
	RETURN;
END_IF

FOR nIndex := 1 TO _Count DO
	IF _Names[nIndex] = sName THEN
		_BaseUnits[nIndex] := BaseUnit;
		M_RegisterReference := TRUE;
		RETURN;
	END_IF
END_FOR

nIndex := _Count + 1;
IF nIndex > Param_Config.MaxConfigReferenceNodes THEN
	Error := TRUE;
	ErrorMessage := 'Reference registry is full.';
	RETURN;
END_IF

_Names[nIndex] := sName;
_BaseUnits[nIndex] := BaseUnit;
_Count := nIndex;
M_RegisterReference := TRUE;
END_METHOD

METHOD PUBLIC M_Resolve : I_BaseUnit
VAR_INPUT
	Name : STRING(255);
END_VAR
VAR
	nIndex : UINT;
END_VAR
M_Resolve := 0;
Error := FALSE;
ErrorMessage := '';
FOR nIndex := 1 TO _Count DO
	IF _Names[nIndex] = Name THEN
		M_Resolve := _BaseUnits[nIndex];
		RETURN;
	END_IF
END_FOR
Error := TRUE;
ErrorMessage := 'Reference source was not registered.';
END_METHOD

END_FUNCTION_BLOCK

// ---- Configuration/POUs/FB_ModuleReferenceBindingContext.TcPOU
FUNCTION_BLOCK FB_ModuleReferenceBindingContext IMPLEMENTS I_ModuleReferenceBindings
VAR_OUTPUT
	Error : BOOL;
	ErrorMessage : STRING(255);
END_VAR
VAR
	_Names : ARRAY[1..Param_Config.MaxModuleReferences] OF STRING(80);
	_SourceNames : ARRAY[1..Param_Config.MaxModuleReferences] OF STRING(255);
	_Consumed : ARRAY[1..Param_Config.MaxModuleReferences] OF BOOL;
	_ReferenceManager : REFERENCE TO FB_ReferenceManager;
	_Count : UINT;
	_Active : BOOL;
END_VAR

METHOD PUBLIC M_Begin : BOOL
VAR_IN_OUT CONSTANT
	ModuleConfig : ST_ModuleFileConfig;
END_VAR
VAR_IN_OUT
	ReferenceManager : FB_ReferenceManager;
END_VAR
VAR
	nItem : UINT;
	nOther : UINT;
END_VAR
M_Begin := FALSE;
M_Clear();

IF ModuleConfig.ReferenceCount > Param_Config.MaxModuleReferences THEN
	Error := TRUE;
	ErrorMessage := 'Module reference capacity was exceeded.';
	RETURN;
END_IF

FOR nItem := 1 TO ModuleConfig.ReferenceCount DO
	IF (ModuleConfig.References[nItem].Name = '') OR (ModuleConfig.References[nItem].Source = '') THEN
		Error := TRUE;
		ErrorMessage := 'Every Module reference requires a name and source.';
		RETURN;
	END_IF

	IF nItem > 1 THEN
		FOR nOther := 1 TO nItem - 1 DO
			IF ModuleConfig.References[nOther].Name = ModuleConfig.References[nItem].Name THEN
				Error := TRUE;
				ErrorMessage := CONCAT('Duplicate Module reference name: ', ModuleConfig.References[nItem].Name);
				RETURN;
			END_IF
		END_FOR
	END_IF

	_Names[nItem] := ModuleConfig.References[nItem].Name;
	_SourceNames[nItem] := ModuleConfig.References[nItem].Source;
END_FOR

_Count := ModuleConfig.ReferenceCount;
_ReferenceManager REF= ReferenceManager;
_Active := TRUE;
M_Begin := TRUE;
END_METHOD

METHOD PUBLIC M_Clear
VAR
	nItem : UINT;
END_VAR
FOR nItem := 1 TO Param_Config.MaxModuleReferences DO
	_Names[nItem] := '';
	_SourceNames[nItem] := '';
	_Consumed[nItem] := FALSE;
END_FOR
_Count := 0;
_Active := FALSE;
Error := FALSE;
ErrorMessage := '';
END_METHOD

METHOD PUBLIC M_End : BOOL
VAR
	nItem : UINT;
END_VAR
M_End := FALSE;
IF Error THEN
	RETURN;
END_IF
IF NOT _Active THEN
	Error := TRUE;
	ErrorMessage := 'No Module reference binding context is active.';
	RETURN;
END_IF

FOR nItem := 1 TO _Count DO
	IF NOT _Consumed[nItem] THEN
		Error := TRUE;
		ErrorMessage := CONCAT('Unknown Module reference name: ', _Names[nItem]);
		RETURN;
	END_IF
END_FOR

_Active := FALSE;
M_End := TRUE;
END_METHOD

METHOD PRIVATE M_Take : I_BaseUnit
VAR_INPUT
	Name : STRING(80);
	Required : BOOL;
END_VAR
VAR_OUTPUT
	Present : BOOL;
	TakeErrorMessage : STRING(255);
END_VAR
VAR
	nItem : UINT;
	BaseUnit : I_BaseUnit;
END_VAR
M_Take := 0;
Present := FALSE;
TakeErrorMessage := '';
IF Error THEN
	TakeErrorMessage := ErrorMessage;
	RETURN;
END_IF
IF NOT _Active THEN
	Error := TRUE;
	ErrorMessage := 'No Module reference binding context is active.';
	TakeErrorMessage := ErrorMessage;
	RETURN;
END_IF
IF Name = '' THEN
	Error := TRUE;
	ErrorMessage := 'A Module reference name is required.';
	TakeErrorMessage := ErrorMessage;
	RETURN;
END_IF

FOR nItem := 1 TO _Count DO
	IF _Names[nItem] = Name THEN
		IF _Consumed[nItem] THEN
			Error := TRUE;
			ErrorMessage := CONCAT('Module reference was taken more than once: ', Name);
			TakeErrorMessage := ErrorMessage;
			RETURN;
		END_IF
		IF NOT __ISVALIDREF(_ReferenceManager) THEN
			Error := TRUE;
			ErrorMessage := 'The Module reference source registry is unavailable.';
			TakeErrorMessage := ErrorMessage;
			RETURN;
		END_IF
		BaseUnit := _ReferenceManager.M_Resolve(Name := _SourceNames[nItem]);
		IF BaseUnit = 0 THEN
			Error := TRUE;
			ErrorMessage := CONCAT('Module reference source was not registered: ', _SourceNames[nItem]);
			TakeErrorMessage := ErrorMessage;
			RETURN;
		END_IF
		_Consumed[nItem] := TRUE;
		Present := TRUE;
		M_Take := BaseUnit;
		RETURN;
	END_IF
END_FOR

IF Required THEN
	Error := TRUE;
	ErrorMessage := CONCAT('Missing required Module reference: ', Name);
	TakeErrorMessage := ErrorMessage;
END_IF
END_METHOD

METHOD PUBLIC M_TakeOptional : I_BaseUnit
VAR_INPUT
	Name : STRING(80);
END_VAR
VAR_OUTPUT
	Present : BOOL;
	ErrorMessage : STRING(255);
END_VAR
M_TakeOptional := M_Take(
	Name := Name,
	Required := FALSE,
	Present => Present,
	TakeErrorMessage => ErrorMessage);
END_METHOD

METHOD PUBLIC M_TakeRequired : I_BaseUnit
VAR_INPUT
	Name : STRING(80);
END_VAR
VAR_OUTPUT
	ErrorMessage : STRING(255);
END_VAR
VAR
	bPresent : BOOL;
END_VAR
M_TakeRequired := M_Take(
	Name := Name,
	Required := TRUE,
	Present => bPresent,
	TakeErrorMessage => ErrorMessage);
END_METHOD

END_FUNCTION_BLOCK

// ---- Configuration/POUs/FB_LinkVariableManager.TcPOU
FUNCTION_BLOCK FB_LinkVariableManager IMPLEMENTS I_VariableNodeReader
VAR_OUTPUT
	Error : BOOL;
	ErrorMessage : STRING(255);
END_VAR
VAR
	_Nodes : ARRAY[1..Param_Config.MaxConfigVariableNodes] OF ST_LinkVariableNode;
	_NodeCount : UINT;
	_InfrastructureNodeCount : UINT;
	_InfrastructureSealed : BOOL;
	_InfrastructureRegistrationActive : BOOL;
	_ModuleRegistrationActive : BOOL;
	_ModuleRootName : STRING(255);
	_ModuleConfig : REFERENCE TO ST_ModuleFileConfig;
	_Links : ARRAY[1..Param_Config.MaxModuleMappings * Param_Config.MaxTotalConfiguredModules * 2] OF ST_VariableLink;
	_LinkCount : UINT;
	_TargetWriterSourceNodes : ARRAY[1..Param_Config.MaxConfigVariableNodes] OF UINT;
	_JsonDataType : FB_JsonReadWriteDataType;
END_VAR

METHOD PUBLIC M_AddLink : BOOL
VAR_INPUT
	SourceName : STRING(255);
	TargetName : STRING(255);
	SourceDataType : E_ConfigDataType;
	TargetDataType : E_ConfigDataType;
	Phase : E_LinkPhase;
	HasTransform : BOOL;
	Scale : LREAL;
	Offset : LREAL;
END_VAR
VAR
	nSource : UINT;
	nTarget : UINT;
	nNext : UINT;
END_VAR
M_AddLink := FALSE;
Error := FALSE;
ErrorMessage := '';

nSource := M_FindNode(Name := SourceName);
nTarget := M_FindNode(Name := TargetName);
IF (nSource = 0) OR (nTarget = 0) THEN
	Error := TRUE;
	ErrorMessage := 'Link source or target was not registered.';
	RETURN;
END_IF

IF _Nodes[nSource].Access = E_VariableAccess.WriteOnly THEN
	Error := TRUE;
	ErrorMessage := 'Link source is write-only.';
	RETURN;
END_IF
IF _Nodes[nTarget].Access = E_VariableAccess.ReadOnly THEN
	Error := TRUE;
	ErrorMessage := 'Link target is read-only.';
	RETURN;
END_IF

IF (SourceDataType <> E_ConfigDataType.Unknown) AND (_Nodes[nSource].DataType <> SourceDataType) THEN
	Error := TRUE;
	ErrorMessage := 'Link source type does not match the registered node.';
	RETURN;
END_IF
IF (TargetDataType <> E_ConfigDataType.Unknown) AND (_Nodes[nTarget].DataType <> TargetDataType) THEN
	Error := TRUE;
	ErrorMessage := 'Link target type does not match the registered node.';
	RETURN;
END_IF

IF HasTransform THEN
	IF NOT M_IsNumeric(DataType := _Nodes[nSource].DataType)
		OR NOT M_IsNumeric(DataType := _Nodes[nTarget].DataType) THEN
		Error := TRUE;
		ErrorMessage := 'scale/offset requires numeric source and target nodes.';
		RETURN;
	END_IF
ELSE
	IF (_Nodes[nSource].DataType <> _Nodes[nTarget].DataType)
		OR (_Nodes[nSource].Size <> _Nodes[nTarget].Size) THEN
		Error := TRUE;
		ErrorMessage := 'MEMCPY links require identical type and size.';
		RETURN;
	END_IF
END_IF

IF _TargetWriterSourceNodes[nTarget] <> 0 THEN
	Error := TRUE;
	ErrorMessage := CONCAT(
		CONCAT('Link target already has a writer: ', TargetName),
		CONCAT(' (existing source: ', CONCAT(_Nodes[_TargetWriterSourceNodes[nTarget]].Name, ').')));
	RETURN;
END_IF

nNext := _LinkCount + 1;
IF nNext > (Param_Config.MaxModuleMappings * Param_Config.MaxTotalConfiguredModules * 2) THEN
	Error := TRUE;
	ErrorMessage := 'Link table is full.';
	RETURN;
END_IF

_Links[nNext].SourceAddress := _Nodes[nSource].Address;
_Links[nNext].TargetAddress := _Nodes[nTarget].Address;
_Links[nNext].SourceSize := _Nodes[nSource].Size;
_Links[nNext].TargetSize := _Nodes[nTarget].Size;
_Links[nNext].SourceDataType := _Nodes[nSource].DataType;
_Links[nNext].TargetDataType := _Nodes[nTarget].DataType;
_Links[nNext].Phase := Phase;
_Links[nNext].HasTransform := HasTransform;
_Links[nNext].Scale := Scale;
_Links[nNext].Offset := Offset;
_LinkCount := nNext;
_TargetWriterSourceNodes[nTarget] := nSource;
M_AddLink := TRUE;
END_METHOD

METHOD PUBLIC M_BeginInfrastructureRegistration : BOOL
VAR
	nIndex : UINT;
END_VAR
M_BeginInfrastructureRegistration := FALSE;
IF _InfrastructureRegistrationActive THEN
	IF NOT Error THEN
		Error := TRUE;
		ErrorMessage := 'An Infrastructure registration session is already active.';
	END_IF
	RETURN;
END_IF
IF _InfrastructureSealed THEN
	IF NOT Error THEN
		Error := TRUE;
		ErrorMessage := 'Infrastructure node registration is already sealed.';
	END_IF
	RETURN;
END_IF
IF _ModuleRegistrationActive THEN
	IF NOT Error THEN
		Error := TRUE;
		ErrorMessage := 'Cannot begin Infrastructure registration during Module registration.';
	END_IF
	RETURN;
END_IF

Error := FALSE;
ErrorMessage := '';
FOR nIndex := 1 TO _NodeCount DO
	MEMSET(ADR(_Nodes[nIndex]), 0, SIZEOF(_Nodes[nIndex]));
END_FOR
_NodeCount := 0;
_InfrastructureNodeCount := 0;
_InfrastructureRegistrationActive := TRUE;
M_BeginInfrastructureRegistration := TRUE;
END_METHOD

METHOD PUBLIC M_BeginModuleRegistration : BOOL
VAR_INPUT
	Address : PVOID;
	Size : UDINT;
END_VAR
VAR_IN_OUT
	ModuleConfig : ST_ModuleFileConfig;
END_VAR
VAR
	hrErrorCode : HRESULT;
END_VAR
M_BeginModuleRegistration := FALSE;
IF _InfrastructureRegistrationActive THEN
	IF NOT Error THEN
		Error := TRUE;
		ErrorMessage := 'Cannot begin Module registration during Infrastructure registration.';
	END_IF
	RETURN;
END_IF
IF _ModuleRegistrationActive THEN
	IF NOT Error THEN
		Error := TRUE;
		ErrorMessage := 'A Module registration session is already active.';
	END_IF
	RETURN;
END_IF
Error := FALSE;
ErrorMessage := '';
_ModuleRegistrationActive := FALSE;
_ModuleRootName := '';

IF NOT _InfrastructureSealed THEN
	Error := TRUE;
	ErrorMessage := 'Infrastructure node registration must be sealed before Module registration.';
	RETURN;
END_IF
IF (Address = 0) OR (Size = 0) THEN
	Error := TRUE;
	ErrorMessage := 'Cannot register a Module without a valid address and size.';
	RETURN;
END_IF

_ModuleRootName := _JsonDataType.GetSymbolNameByAddress(
	nData := Size,
	pData := Address,
	hrErrorCode => hrErrorCode);
IF (hrErrorCode <> 0) OR (_ModuleRootName = '') THEN
	Error := TRUE;
	ErrorMessage := 'Cannot resolve the Module ADS symbol name.';
	RETURN;
END_IF

_ModuleConfig REF=ModuleConfig;
_ModuleRegistrationActive := TRUE;
M_BeginModuleRegistration := TRUE;
END_METHOD

METHOD PRIVATE M_BuildNodeName : BOOL
VAR_INPUT
	RootName : STRING(255);
	RelativeName : STRING(255);
END_VAR
VAR_OUTPUT
	FullName : STRING(255);
END_VAR
M_BuildNodeName := FALSE;
FullName := '';

IF RootName = '' THEN
	Error := TRUE;
	ErrorMessage := 'Cannot register nodes without a root symbol name.';
	RETURN;
END_IF
IF (LEN(RootName) + LEN(RelativeName) + 1) > 255 THEN
	Error := TRUE;
	ErrorMessage := 'Registered node symbol name exceeds 255 characters.';
	RETURN;
END_IF

FullName := CONCAT(CONCAT(RootName,'.'), RelativeName);
M_BuildNodeName := TRUE;
END_METHOD

METHOD PUBLIC M_ClearLinks
MEMSET(ADR(_Links), 0, SIZEOF(_Links));
MEMSET(ADR(_TargetWriterSourceNodes), 0, SIZEOF(_TargetWriterSourceNodes));
_LinkCount := 0;
Error := FALSE;
ErrorMessage := '';
END_METHOD

METHOD PUBLIC M_ClearModuleNodes
VAR
	nIndex : UINT;
END_VAR
IF _InfrastructureSealed THEN
	FOR nIndex := _InfrastructureNodeCount + 1 TO _NodeCount DO
		MEMSET(ADR(_Nodes[nIndex]), 0, SIZEOF(_Nodes[nIndex]));
	END_FOR
	_NodeCount := _InfrastructureNodeCount;
END_IF
_ModuleRegistrationActive := FALSE;
_ModuleRootName := '';
Error := FALSE;
ErrorMessage := '';
END_METHOD

METHOD PRIVATE M_CopyPhase
VAR_INPUT
	Phase : E_LinkPhase;
END_VAR
VAR
	nIndex : UINT;
	fSource : LREAL;
	bValid : BOOL;
END_VAR
FOR nIndex := 1 TO _LinkCount DO
	IF _Links[nIndex].Phase <> Phase THEN
		CONTINUE;
	END_IF

	IF _Links[nIndex].HasTransform THEN
		fSource := M_ReadNumeric(
			Address := _Links[nIndex].SourceAddress,
			DataType := _Links[nIndex].SourceDataType,
			Valid => bValid);
		IF bValid THEN
			M_WriteNumeric(
				Address := _Links[nIndex].TargetAddress,
				DataType := _Links[nIndex].TargetDataType,
				Value := (fSource * _Links[nIndex].Scale) + _Links[nIndex].Offset);
		END_IF
	ELSE
		MEMCPY(
			destAddr := _Links[nIndex].TargetAddress,
			srcAddr := _Links[nIndex].SourceAddress,
			n := _Links[nIndex].SourceSize);
	END_IF
END_FOR
END_METHOD

METHOD PUBLIC M_CyclicInput
M_CopyPhase(Phase := E_LinkPhase.InputToModule);
END_METHOD

METHOD PUBLIC M_CyclicOutput
M_CopyPhase(Phase := E_LinkPhase.ModuleToOutput);
END_METHOD

METHOD PUBLIC M_EndModuleRegistration : BOOL
VAR_OUTPUT
	ModuleSymbol : STRING(255);
END_VAR
VAR
	nItem : UINT;
END_VAR
M_EndModuleRegistration := FALSE;
ModuleSymbol := '';
IF Error THEN
	_ModuleRegistrationActive := FALSE;
	RETURN;
END_IF
IF NOT _ModuleRegistrationActive OR NOT __ISVALIDREF(_ModuleConfig) THEN
	Error := TRUE;
	ErrorMessage := 'No Module registration session is active.';
	RETURN;
END_IF

FOR nItem := 1 TO _ModuleConfig.InputMappingCount DO
	IF NOT M_RequireRelativeNode(RelativeName := _ModuleConfig.InputMappings[nItem].Target) THEN
		_ModuleRegistrationActive := FALSE;
		RETURN;
	END_IF
END_FOR
FOR nItem := 1 TO _ModuleConfig.OutputMappingCount DO
	IF NOT M_RequireRelativeNode(RelativeName := _ModuleConfig.OutputMappings[nItem].Source) THEN
		_ModuleRegistrationActive := FALSE;
		RETURN;
	END_IF
END_FOR
FOR nItem := 1 TO _ModuleConfig.VariableCount DO
	IF NOT M_RequireRelativeNode(RelativeName := _ModuleConfig.VariableList[nItem].Source) THEN
		_ModuleRegistrationActive := FALSE;
		RETURN;
	END_IF
END_FOR
FOR nItem := 1 TO _ModuleConfig.AlarmCount DO
	IF NOT M_RequireRelativeNode(RelativeName := _ModuleConfig.AlarmList[nItem].Source) THEN
		_ModuleRegistrationActive := FALSE;
		RETURN;
	END_IF
END_FOR

ModuleSymbol := _ModuleRootName;
_ModuleRegistrationActive := FALSE;
M_EndModuleRegistration := TRUE;
END_METHOD

METHOD PRIVATE M_FindNode : UINT
VAR_INPUT
	Name : STRING(255);
END_VAR
VAR
	nIndex : UINT;
END_VAR
M_FindNode := 0;
FOR nIndex := 1 TO _NodeCount DO
	IF _Nodes[nIndex].Name = Name THEN
		M_FindNode := nIndex;
		RETURN;
	END_IF
END_FOR
END_METHOD

METHOD PRIVATE M_IsNumeric : BOOL
VAR_INPUT
	DataType : E_ConfigDataType;
END_VAR
M_IsNumeric := (DataType = E_ConfigDataType.Integer32)
	OR (DataType = E_ConfigDataType.UnsignedInteger32)
	OR (DataType = E_ConfigDataType.Float32)
	OR (DataType = E_ConfigDataType.Float64);
END_METHOD

METHOD PUBLIC M_ReadNode : BOOL
VAR_INPUT
	NodeHandle : UINT;
	ExpectedDataType : E_ConfigDataType;
END_VAR
VAR_IN_OUT
	Value : ST_ConfigRawValue;
END_VAR
VAR_OUTPUT
	ErrorCode : E_ConfigValueError;
END_VAR
M_ReadNode := FALSE;
ErrorCode := E_ConfigValueError.None;
MEMSET(ADR(Value), 0, SIZEOF(Value));

IF (NodeHandle < 1) OR (NodeHandle > _NodeCount) THEN
	ErrorCode := E_ConfigValueError.InvalidNodeHandle;
	RETURN;
END_IF
IF _Nodes[NodeHandle].Access = E_VariableAccess.WriteOnly THEN
	ErrorCode := E_ConfigValueError.NodeReadNotAllowed;
	RETURN;
END_IF
IF _Nodes[NodeHandle].Address = 0 THEN
	ErrorCode := E_ConfigValueError.InvalidNodeAddress;
	RETURN;
END_IF
IF (ExpectedDataType = E_ConfigDataType.Unknown)
	OR (_Nodes[NodeHandle].DataType <> ExpectedDataType) THEN
	ErrorCode := E_ConfigValueError.NodeDataTypeMismatch;
	RETURN;
END_IF
IF (_Nodes[NodeHandle].Size = 0)
	OR (_Nodes[NodeHandle].Size > SIZEOF(Value.Data)) THEN
	ErrorCode := E_ConfigValueError.InvalidNodeSize;
	RETURN;
END_IF

MEMCPY(
	destAddr := ADR(Value.Data),
	srcAddr := _Nodes[NodeHandle].Address,
	n := _Nodes[NodeHandle].Size);
M_ReadNode := TRUE;
END_METHOD

METHOD PRIVATE M_ReadNumeric : LREAL
VAR_INPUT
	Address : PVOID;
	DataType : E_ConfigDataType;
END_VAR
VAR_OUTPUT
	Valid : BOOL;
END_VAR
VAR
	pDInt : POINTER TO DINT;
	pUDInt : POINTER TO UDINT;
	pReal : POINTER TO REAL;
	pLReal : POINTER TO LREAL;
END_VAR
Valid := TRUE;
CASE DataType OF
	E_ConfigDataType.Integer32:
		pDInt := Address;
		M_ReadNumeric := DINT_TO_LREAL(pDInt^);
	E_ConfigDataType.UnsignedInteger32:
		pUDInt := Address;
		M_ReadNumeric := UDINT_TO_LREAL(pUDInt^);
	E_ConfigDataType.Float32:
		pReal := Address;
		M_ReadNumeric := REAL_TO_LREAL(pReal^);
	E_ConfigDataType.Float64:
		pLReal := Address;
		M_ReadNumeric := pLReal^;
ELSE
	Valid := FALSE;
	M_ReadNumeric := 0.0;
END_CASE
END_METHOD

METHOD PUBLIC M_RegisterInfrastructureNode : BOOL
VAR_INPUT
	Variable : ANY;
	Access : E_VariableAccess;
END_VAR
VAR
	sNodeName : STRING(255);
	hrErrorCode : HRESULT;
END_VAR
M_RegisterInfrastructureNode := FALSE;
IF Error THEN
	RETURN;
END_IF
IF NOT _InfrastructureRegistrationActive THEN
	Error := TRUE;
	ErrorMessage := 'No Infrastructure registration session is active.';
	RETURN;
END_IF
IF _InfrastructureSealed THEN
	Error := TRUE;
	ErrorMessage := 'Infrastructure node registration is already sealed.';
	RETURN;
END_IF
IF (Variable.pValue = 0) OR (Variable.diSize <= 0) THEN
	Error := TRUE;
	ErrorMessage := 'An Infrastructure node requires a valid address and positive size.';
	RETURN;
END_IF
IF (Access <> E_VariableAccess.ReadOnly)
	AND (Access <> E_VariableAccess.WriteOnly)
	AND (Access <> E_VariableAccess.ReadWrite) THEN
	Error := TRUE;
	ErrorMessage := 'Registered node access is invalid.';
	RETURN;
END_IF

sNodeName := _JsonDataType.GetSymbolNameByAddress(
	nData := DINT_TO_UDINT(Variable.diSize),
	pData := Variable.pValue,
	hrErrorCode => hrErrorCode);
IF (hrErrorCode <> 0) OR (sNodeName = '') THEN
	Error := TRUE;
	ErrorMessage := 'Cannot resolve the Infrastructure node ADS symbol name.';
	RETURN;
END_IF

IF M_FindNode(Name := sNodeName) <> 0 THEN
	Error := TRUE;
	ErrorMessage := CONCAT('Duplicate Infrastructure node declaration: ', sNodeName);
	RETURN;
END_IF
M_RegisterInfrastructureNode := M_RegisterNode(
	Name := sNodeName,
	Variable := Variable,
	Access := Access);
END_METHOD

METHOD PRIVATE M_RegisterNode : BOOL
VAR_INPUT
	Name : STRING(255);
	Variable : ANY;
	Access : E_VariableAccess;
END_VAR
VAR
	nIndex : UINT;
	eDataType : E_ConfigDataType;
END_VAR
M_RegisterNode := FALSE;
IF Error THEN
	RETURN;
END_IF
IF (Name = '') OR (Variable.pValue = 0) OR (Variable.diSize <= 0) THEN
	Error := TRUE;
	ErrorMessage := 'Registered node requires a name, address and positive size.';
	RETURN;
END_IF
IF (Access <> E_VariableAccess.ReadOnly)
	AND (Access <> E_VariableAccess.WriteOnly)
	AND (Access <> E_VariableAccess.ReadWrite) THEN
	Error := TRUE;
	ErrorMessage := 'Registered node access is invalid.';
	RETURN;
END_IF

CASE Variable.TypeClass OF
	__SYSTEM.TYPE_CLASS.TYPE_BOOL:
		eDataType := E_ConfigDataType.Boolean;
	__SYSTEM.TYPE_CLASS.TYPE_DINT:
		eDataType := E_ConfigDataType.Integer32;
	__SYSTEM.TYPE_CLASS.TYPE_UDINT:
		eDataType := E_ConfigDataType.UnsignedInteger32;
	__SYSTEM.TYPE_CLASS.TYPE_REAL:
		eDataType := E_ConfigDataType.Float32;
	__SYSTEM.TYPE_CLASS.TYPE_LREAL:
		eDataType := E_ConfigDataType.Float64;
	__SYSTEM.TYPE_CLASS.TYPE_STRING:
		eDataType := E_ConfigDataType.String80;
ELSE
	Error := TRUE;
	ErrorMessage := 'Only BOOL, DINT, UDINT, REAL, LREAL and STRING nodes are supported.';
	RETURN;
END_CASE

IF (eDataType <> E_ConfigDataType.String80)
	AND (DINT_TO_UDINT(Variable.diSize) <> F_ConfigDataTypeSize(DataType := eDataType)) THEN
	Error := TRUE;
	ErrorMessage := 'Registered node size does not match its primitive type.';
	RETURN;
END_IF
IF (eDataType = E_ConfigDataType.String80) AND (Variable.diSize > Param_Config.MaxConfigValueSize) THEN
	Error := TRUE;
	ErrorMessage := 'Registered STRING exceeds STRING(80).';
	RETURN;
END_IF

nIndex := M_FindNode(Name := Name);
IF nIndex = 0 THEN
	nIndex := _NodeCount + 1;
	IF nIndex > Param_Config.MaxConfigVariableNodes THEN
		Error := TRUE;
		ErrorMessage := 'Variable node registry is full.';
		RETURN;
	END_IF
	_NodeCount := nIndex;
END_IF

_Nodes[nIndex].Name := Name;
_Nodes[nIndex].Address := Variable.pValue;
_Nodes[nIndex].Size := DINT_TO_UDINT(Variable.diSize);
_Nodes[nIndex].DataType := eDataType;
_Nodes[nIndex].Access := Access;
M_RegisterNode := TRUE;
END_METHOD

METHOD PUBLIC M_RegisterModuleNode : BOOL
VAR_INPUT
	Variable : ANY;
	Access : E_VariableAccess;
END_VAR
VAR
	sNodeName : STRING(255);
	sModulePrefix : STRING(255);
	hrErrorCode : HRESULT;
END_VAR
M_RegisterModuleNode := FALSE;
IF Error THEN
	RETURN;
END_IF
IF NOT _ModuleRegistrationActive THEN
	Error := TRUE;
	ErrorMessage := 'No Module registration session is active.';
	RETURN;
END_IF
IF (Variable.pValue = 0) OR (Variable.diSize <= 0) THEN
	Error := TRUE;
	ErrorMessage := 'A Module node requires a valid address and positive size.';
	RETURN;
END_IF

sNodeName := _JsonDataType.GetSymbolNameByAddress(
	nData := DINT_TO_UDINT(Variable.diSize),
	pData := Variable.pValue,
	hrErrorCode => hrErrorCode);
IF (hrErrorCode <> 0) OR (sNodeName = '') THEN
	Error := TRUE;
	ErrorMessage := 'Cannot resolve the Module node ADS symbol name.';
	RETURN;
END_IF

sModulePrefix := CONCAT(_ModuleRootName, '.');
IF LEFT(sNodeName, LEN(sModulePrefix)) <> sModulePrefix THEN
	Error := TRUE;
	ErrorMessage := 'The registered node does not belong to the active Module instance.';
	RETURN;
END_IF

IF M_FindNode(Name := sNodeName) <> 0 THEN
	Error := TRUE;
	ErrorMessage := CONCAT('Duplicate Module node declaration: ', sNodeName);
	RETURN;
END_IF
M_RegisterModuleNode := M_RegisterNode(Name := sNodeName, Variable := Variable, Access := Access);
END_METHOD

METHOD PRIVATE M_RequireRelativeNode : BOOL
VAR_INPUT
	RelativeName : STRING(255);
END_VAR
VAR
	sNodeName : STRING(255);
END_VAR
M_RequireRelativeNode := FALSE;
IF NOT M_BuildNodeName(
	RootName := _ModuleRootName,
	RelativeName := RelativeName,
	FullName => sNodeName) THEN
	RETURN;
END_IF
IF M_FindNode(Name := sNodeName) = 0 THEN
	Error := TRUE;
	ErrorMessage := CONCAT('Module node was not declared by its adapter: ', RelativeName);
	RETURN;
END_IF
M_RequireRelativeNode := TRUE;
END_METHOD

METHOD PUBLIC M_ResolveReadableNode : BOOL
VAR_INPUT
	Name : STRING(255);
	ExpectedDataType : E_ConfigDataType;
END_VAR
VAR_OUTPUT
	NodeHandle : UINT;
END_VAR
VAR
	nNode : UINT;
END_VAR
M_ResolveReadableNode := FALSE;
NodeHandle := 0;
Error := FALSE;
ErrorMessage := '';

nNode := M_FindNode(Name := Name);
IF nNode = 0 THEN
	Error := TRUE;
	ErrorMessage := CONCAT('Configured value source was not registered: ', Name);
	RETURN;
END_IF
IF _Nodes[nNode].Access = E_VariableAccess.WriteOnly THEN
	Error := TRUE;
	ErrorMessage := CONCAT('Configured value source is write-only: ', Name);
	RETURN;
END_IF
IF _Nodes[nNode].Address = 0 THEN
	Error := TRUE;
	ErrorMessage := CONCAT('Configured value source has no valid address: ', Name);
	RETURN;
END_IF
IF (ExpectedDataType = E_ConfigDataType.Unknown)
	OR (_Nodes[nNode].DataType <> ExpectedDataType) THEN
	Error := TRUE;
	ErrorMessage := CONCAT('Configured value source type does not match the registered node: ', Name);
	RETURN;
END_IF
IF (_Nodes[nNode].Size = 0)
	OR (_Nodes[nNode].Size > Param_Config.MaxConfigValueSize) THEN
	Error := TRUE;
	ErrorMessage := CONCAT('Configured value source size is unsupported: ', Name);
	RETURN;
END_IF

NodeHandle := nNode;
M_ResolveReadableNode := TRUE;
END_METHOD

METHOD PUBLIC M_SealInfrastructureRegistration : BOOL
VAR
	nIndex : UINT;
END_VAR
M_SealInfrastructureRegistration := FALSE;
IF Error THEN
	IF _InfrastructureRegistrationActive THEN
		FOR nIndex := 1 TO _NodeCount DO
			MEMSET(ADR(_Nodes[nIndex]), 0, SIZEOF(_Nodes[nIndex]));
		END_FOR
		_NodeCount := 0;
		_InfrastructureNodeCount := 0;
		_InfrastructureRegistrationActive := FALSE;
	END_IF
	RETURN;
END_IF
IF NOT _InfrastructureRegistrationActive THEN
	Error := TRUE;
	ErrorMessage := 'No Infrastructure registration session is active.';
	RETURN;
END_IF
IF _ModuleRegistrationActive THEN
	Error := TRUE;
	ErrorMessage := 'Cannot seal infrastructure nodes during Module registration.';
	FOR nIndex := 1 TO _NodeCount DO
		MEMSET(ADR(_Nodes[nIndex]), 0, SIZEOF(_Nodes[nIndex]));
	END_FOR
	_NodeCount := 0;
	_InfrastructureNodeCount := 0;
	_InfrastructureRegistrationActive := FALSE;
	RETURN;
END_IF
_InfrastructureNodeCount := _NodeCount;
_InfrastructureSealed := TRUE;
_InfrastructureRegistrationActive := FALSE;
M_SealInfrastructureRegistration := TRUE;
END_METHOD

METHOD PRIVATE M_WriteNumeric
VAR_INPUT
	Address : PVOID;
	DataType : E_ConfigDataType;
	Value : LREAL;
END_VAR
VAR
	pDInt : POINTER TO DINT;
	pUDInt : POINTER TO UDINT;
	pReal : POINTER TO REAL;
	pLReal : POINTER TO LREAL;
END_VAR
CASE DataType OF
	E_ConfigDataType.Integer32:
		pDInt := Address;
		pDInt^ := LREAL_TO_DINT(Value);
	E_ConfigDataType.UnsignedInteger32:
		pUDInt := Address;
		pUDInt^ := LREAL_TO_UDINT(Value);
	E_ConfigDataType.Float32:
		pReal := Address;
		pReal^ := LREAL_TO_REAL(Value);
	E_ConfigDataType.Float64:
		pLReal := Address;
		pLReal^ := Value;
END_CASE
END_METHOD

END_FUNCTION_BLOCK

// ---- Configuration/POUs/FB_ModuleConfigurationManager.TcPOU
FUNCTION_BLOCK FB_ModuleConfigurationManager
VAR_INPUT
	Execute : BOOL;
	FilePath : STRING(255);
END_VAR
VAR_IN_OUT
	LinkVariableManager : FB_LinkVariableManager;
	ReferenceManager : FB_ReferenceManager;
	ModuleTypeRegistry : FB_ModuleTypeRegistry;
END_VAR
VAR_OUTPUT
	Ready : BOOL;
	Busy : BOOL;
	Error : BOOL;
	ErrorCode : HRESULT;
	ErrorMessage : STRING(255);
END_VAR
VAR
	_Json : FB_JsonDomParser;
	_Config : ST_SystemFileConfig;
	_bLoad : BOOL;
	_bLoaded : BOOL;
	_nState : USINT;
	_nRevision : UDINT;
	_RuntimeConfigScratch : ST_ModuleRuntimeConfig;
	_ReferenceBindingContext : FB_ModuleReferenceBindingContext;
END_VAR

CASE _nState OF
	0:
		Busy := FALSE;
		IF Execute THEN
			Ready := FALSE;
			Error := FALSE;
			ErrorCode := 0;
			ErrorMessage := '';
			_bLoad := TRUE;
			Busy := TRUE;
			_nState := 1;
		END_IF

	1:
		Busy := TRUE;
		_bLoaded := _Json.LoadDocumentFromFile(
			sFile := FilePath,
			bExec := _bLoad,
			hrErrorCode => ErrorCode);
		IF _bLoaded THEN
			IF M_ParseDocument() THEN
				_nState := 2;
			ELSE
				Error := TRUE;
				M_ClearAppliedConfiguration(
					LinkVariableManager := LinkVariableManager,
					ModuleTypeRegistry := ModuleTypeRegistry);
				_nState := 3;
			END_IF
		ELSIF NOT _bLoad THEN
			Error := TRUE;
			ErrorMessage := 'Unable to load the UTF-8 JSON module configuration file.';
			M_ClearAppliedConfiguration(
				LinkVariableManager := LinkVariableManager,
				ModuleTypeRegistry := ModuleTypeRegistry);
			_nState := 3;
		END_IF

	2:
		Busy := TRUE;
		IF M_ApplyConfiguration(
			LinkVariableManager := LinkVariableManager,
			ReferenceManager := ReferenceManager,
			ModuleTypeRegistry := ModuleTypeRegistry) THEN
			Ready := TRUE;
		ELSE
			Error := TRUE;
			M_ClearAppliedConfiguration(
				LinkVariableManager := LinkVariableManager,
				ModuleTypeRegistry := ModuleTypeRegistry);
		END_IF
		_nState := 3;

	3:
		Busy := FALSE;
		IF NOT Execute THEN
			_nState := 0;
		END_IF
END_CASE

METHOD PRIVATE M_ApplyConfiguration : BOOL
VAR_IN_OUT
	LinkVariableManager : FB_LinkVariableManager;
	ReferenceManager : FB_ReferenceManager;
	ModuleTypeRegistry : FB_ModuleTypeRegistry;
END_VAR
VAR
	nModule : UINT;
	nOther : UINT;
	nItem : UINT;
	nSlot : UINT;
	sModuleSymbol : STRING(255);
	sFullName : STRING(255);
	Adapter : I_ModuleConfigurationAdapter;
	ReferenceBindings : I_ModuleReferenceBindings;
	sAdapterError : STRING(255);
END_VAR
M_ApplyConfiguration := FALSE;

// Resolve every configured type and reject ambiguous addressing before mutating runtime state.
FOR nModule := 1 TO _Config.ModuleCount DO

	// Check module slot is in range
	IF (_Config.Modules[nModule].Slot < 1)
		OR (_Config.Modules[nModule].Slot > Param_Config.MaxModulePerType) THEN
		ErrorMessage := CONCAT(
			CONCAT('A module slot is outside the supported range 1..', TO_STRING(Param_Config.MaxModulePerType)),
			'.');
		RETURN;
	END_IF

	// Get adapter according to module type
	Adapter := ModuleTypeRegistry.M_Resolve(ModuleTypeName := _Config.Modules[nModule].ModuleType);
	IF Adapter = 0 THEN
		ErrorMessage := ModuleTypeRegistry.ErrorMessage;
		RETURN;
	END_IF

	// Check module slot is supported by specific module (現在各module的slot數量參數共用，其實沒必要檢查)
	IF NOT Adapter.M_IsSlotSupported(Slot := _Config.Modules[nModule].Slot) THEN
		ErrorMessage := 'Module adapter does not support the configured slot.';
		RETURN;
	END_IF

	// Check module id is valid
	IF _Config.Modules[nModule].Enabled THEN
		IF _Config.Modules[nModule].Id = 0 THEN
			ErrorMessage := 'Every enabled module requires a non-zero id.';
			RETURN;
		END_IF
	END_IF

	// Check if module slot/id is duplicate
	FOR nOther := nModule + 1 TO _Config.ModuleCount DO
		IF (_Config.Modules[nModule].ModuleType = _Config.Modules[nOther].ModuleType)
			AND (_Config.Modules[nModule].Slot = _Config.Modules[nOther].Slot) THEN
			ErrorMessage := 'Duplicate module slot for the same module type.';
			RETURN;
		END_IF
		IF _Config.Modules[nModule].Enabled AND _Config.Modules[nOther].Enabled
			AND (_Config.Modules[nModule].Id = _Config.Modules[nOther].Id) THEN
			ErrorMessage := 'Duplicate enabled module ID in configuration.';
			RETURN;
		END_IF
	END_FOR
END_FOR

// 清除 module node & link 資料 (未來要支援 Online Change時這邊才有用)
M_ClearAppliedConfiguration(
	LinkVariableManager := LinkVariableManager,
	ModuleTypeRegistry := ModuleTypeRegistry);

// 記錄重新 Apply 幾次 Configuration (未來要支援 Online Change時這邊才有用)
_nRevision := _nRevision + 1;
IF _nRevision = 0 THEN
	_nRevision := 1;
END_IF


FOR nModule := 1 TO _Config.ModuleCount DO
	nSlot := _Config.Modules[nModule].Slot;

	// Get adapter according to module type
	Adapter := ModuleTypeRegistry.M_Resolve(ModuleTypeName := _Config.Modules[nModule].ModuleType);
	IF Adapter = 0 THEN
		ErrorMessage := ModuleTypeRegistry.ErrorMessage;
		RETURN;
	END_IF

	// Setup runtime config of each module
	MEMSET(ADR(_RuntimeConfigScratch), 0, SIZEOF(_RuntimeConfigScratch));
	_RuntimeConfigScratch.Enabled := _Config.Modules[nModule].Enabled;
	_RuntimeConfigScratch.ModuleId := _Config.Modules[nModule].Id;
	_RuntimeConfigScratch.ModuleType := _Config.Modules[nModule].ModuleType;
	_RuntimeConfigScratch.Revision := _nRevision;

	// Assign runtime config to disable module
	IF NOT _Config.Modules[nModule].Enabled THEN
		_RuntimeConfigScratch.Valid := TRUE;
		IF NOT Adapter.M_ApplyRuntimeConfig(
			Slot := nSlot,
			RuntimeConfig := _RuntimeConfigScratch,
			ErrorMessage => sAdapterError) THEN
			ErrorMessage := sAdapterError;
			RETURN;
		END_IF
		CONTINUE;
	END_IF

	// Initialize the semantic reference map before the adapter pulls its typed bindings.
	// Dictionary of source base unit (from ReferenceManager) & target base unit name (from config file)
	IF NOT _ReferenceBindingContext.M_Begin(
		ModuleConfig := _Config.Modules[nModule],
		ReferenceManager := ReferenceManager) THEN
		ErrorMessage := _ReferenceBindingContext.ErrorMessage;
		RETURN;
	END_IF
	ReferenceBindings := _ReferenceBindingContext;

	// Setup module link variable node & reference binding
	IF NOT Adapter.M_PrepareInstance(
		Slot := nSlot,
		ReferenceBindings := ReferenceBindings,
		ModuleConfig := _Config.Modules[nModule],
		LinkVariableManager := LinkVariableManager,
		ModuleSymbol => sModuleSymbol,
		ErrorMessage => sAdapterError) THEN
		ErrorMessage := sAdapterError;
		RETURN;
	END_IF
	IF NOT _ReferenceBindingContext.M_End() THEN
		ErrorMessage := _ReferenceBindingContext.ErrorMessage;
		RETURN;
	END_IF

	// Build module hardware input link
	FOR nItem := 1 TO _Config.Modules[nModule].InputMappingCount DO
		sFullName := CONCAT(CONCAT(sModuleSymbol, '.'), _Config.Modules[nModule].InputMappings[nItem].Target);
		IF NOT LinkVariableManager.M_AddLink(
			SourceName := _Config.Modules[nModule].InputMappings[nItem].Source,
			TargetName := sFullName,
			SourceDataType := _Config.Modules[nModule].InputMappings[nItem].SourceDataType,
			TargetDataType := _Config.Modules[nModule].InputMappings[nItem].TargetDataType,
			Phase := E_LinkPhase.InputToModule,
			HasTransform := _Config.Modules[nModule].InputMappings[nItem].HasTransform,
			Scale := _Config.Modules[nModule].InputMappings[nItem].Scale,
			Offset := _Config.Modules[nModule].InputMappings[nItem].Offset) THEN
			ErrorMessage := LinkVariableManager.ErrorMessage;
			RETURN;
		END_IF
	END_FOR

	// Build module hardware output link
	FOR nItem := 1 TO _Config.Modules[nModule].OutputMappingCount DO
		sFullName := CONCAT(CONCAT(sModuleSymbol, '.'), _Config.Modules[nModule].OutputMappings[nItem].Source);
		IF NOT LinkVariableManager.M_AddLink(
			SourceName := sFullName,
			TargetName := _Config.Modules[nModule].OutputMappings[nItem].Target,
			SourceDataType := _Config.Modules[nModule].OutputMappings[nItem].SourceDataType,
			TargetDataType := _Config.Modules[nModule].OutputMappings[nItem].TargetDataType,
			Phase := E_LinkPhase.ModuleToOutput,
			HasTransform := _Config.Modules[nModule].OutputMappings[nItem].HasTransform,
			Scale := _Config.Modules[nModule].OutputMappings[nItem].Scale,
			Offset := _Config.Modules[nModule].OutputMappings[nItem].Offset) THEN
			ErrorMessage := LinkVariableManager.ErrorMessage;
			RETURN;
		END_IF
	END_FOR

	// Build module variable list
	_RuntimeConfigScratch.VariableCount := _Config.Modules[nModule].VariableCount;
	FOR nItem := 1 TO _Config.Modules[nModule].VariableCount DO

		// Setup runtime config
		_RuntimeConfigScratch.VariableBindings[nItem].Definition := _Config.Modules[nModule].VariableList[nItem];
		_RuntimeConfigScratch.VariableBindings[nItem].Definition.Source := CONCAT(
			CONCAT(sModuleSymbol, '.'),
			_Config.Modules[nModule].VariableList[nItem].Source);

		// Try resolve node handle by source name and expected data type
		IF NOT LinkVariableManager.M_ResolveReadableNode(
			Name := _RuntimeConfigScratch.VariableBindings[nItem].Definition.Source,
			ExpectedDataType := _RuntimeConfigScratch.VariableBindings[nItem].Definition.DataType,
			NodeHandle => _RuntimeConfigScratch.VariableBindings[nItem].NodeHandle) THEN
			ErrorMessage := LinkVariableManager.ErrorMessage;
			RETURN;
		END_IF
	END_FOR

	// Build module alarm list
	_RuntimeConfigScratch.AlarmCount := _Config.Modules[nModule].AlarmCount;
	FOR nItem := 1 TO _Config.Modules[nModule].AlarmCount DO

		// Setup runtime config
		_RuntimeConfigScratch.AlarmBindings[nItem].Definition := _Config.Modules[nModule].AlarmList[nItem];
		_RuntimeConfigScratch.AlarmBindings[nItem].Definition.Source := CONCAT(
			CONCAT(sModuleSymbol, '.'),
			_Config.Modules[nModule].AlarmList[nItem].Source);

		// Try resolve node handle by source name and expected data type
		IF NOT LinkVariableManager.M_ResolveReadableNode(
			Name := _RuntimeConfigScratch.AlarmBindings[nItem].Definition.Source,
			ExpectedDataType := _RuntimeConfigScratch.AlarmBindings[nItem].Definition.DataType,
			NodeHandle => _RuntimeConfigScratch.AlarmBindings[nItem].NodeHandle) THEN
			ErrorMessage := LinkVariableManager.ErrorMessage;
			RETURN;
		END_IF
	END_FOR

	// Assign runtime config to enable module
	_RuntimeConfigScratch.Valid := TRUE;
	IF NOT Adapter.M_ApplyRuntimeConfig(
		Slot := nSlot,
		RuntimeConfig := _RuntimeConfigScratch,
		ErrorMessage => sAdapterError) THEN
		ErrorMessage := sAdapterError;
		RETURN;
	END_IF
END_FOR

M_ApplyConfiguration := TRUE;
END_METHOD

METHOD PRIVATE M_ClearAppliedConfiguration
VAR_IN_OUT
	LinkVariableManager : FB_LinkVariableManager;
	ModuleTypeRegistry : FB_ModuleTypeRegistry;
END_VAR
LinkVariableManager.M_ClearLinks();
LinkVariableManager.M_ClearModuleNodes();
_ReferenceBindingContext.M_Clear();
ModuleTypeRegistry.M_ClearAll();
END_METHOD

METHOD PRIVATE M_ParseDataType : E_ConfigDataType
VAR_INPUT
	Value : STRING(255);
END_VAR
IF (Value = 'BOOL') OR (Value = 'Bool') OR (Value = 'Boolean') THEN
	M_ParseDataType := E_ConfigDataType.Boolean;
ELSIF (Value = 'DINT') OR (Value = 'DInt') OR (Value = 'Integer_32bit') THEN
	M_ParseDataType := E_ConfigDataType.Integer32;
ELSIF (Value = 'UDINT') OR (Value = 'UDInt') OR (Value = 'Unsigned_32bit') THEN
	M_ParseDataType := E_ConfigDataType.UnsignedInteger32;
ELSIF (Value = 'REAL') OR (Value = 'Real') OR (Value = 'Float_32bit') THEN
	M_ParseDataType := E_ConfigDataType.Float32;
ELSIF (Value = 'LREAL') OR (Value = 'LReal') OR (Value = 'Float_64bit') THEN
	M_ParseDataType := E_ConfigDataType.Float64;
ELSIF (Value = 'STRING') OR (Value = 'String80') OR (Value = 'String_80byte') THEN
	M_ParseDataType := E_ConfigDataType.String80;
ELSE
	M_ParseDataType := E_ConfigDataType.Unknown;
END_IF
END_METHOD

METHOD PRIVATE M_ParseDocument : BOOL
VAR
	Root : SJsonValue;
	Node : SJsonValue;
	ModulesNode : SJsonValue;
	ModuleNode : SJsonValue;
	ArrayNode : SJsonValue;
	ItemNode : SJsonValue;
	TransformNode : SJsonValue;
	ConditionNode : SJsonValue;
	ReferencesNode : SJsonValue;
	ReferenceIterator : SJsonIterator;
	ReferenceIteratorEnd : SJsonIterator;
	nModule : UINT;
	nItem : UINT;
	nOther : UINT;
	nCount : UDINT;
	sValue : STRING(255);
END_VAR
M_ParseDocument := FALSE;
MEMSET(ADR(_Config), 0, SIZEOF(_Config));
Root := _Json.GetDocumentRoot();
IF Root = 0 THEN
	ErrorMessage := 'JSON document has no root object.';
	RETURN;
END_IF

Node := _Json.FindMember(Root, 'schemaVersion');
IF Node = 0 THEN
	ErrorMessage := 'schemaVersion is required.';
	RETURN;
END_IF
_Config.SchemaVersion := _Json.GetUint(Node);
IF _Config.SchemaVersion <> Param_Config.ConfigSchemaVersion THEN
	ErrorMessage := 'Unsupported module configuration schemaVersion.';
	RETURN;
END_IF

Node := _Json.FindMember(Root, 'adsPort');
IF Node <> 0 THEN
	ErrorMessage := 'adsPort is not supported by schemaVersion 4; configured values use registered local nodes.';
	RETURN;
END_IF

ModulesNode := _Json.FindMember(Root, 'modules');
IF (ModulesNode = 0) OR NOT _Json.IsArray(ModulesNode) THEN
	ErrorMessage := 'modules must be a JSON array.';
	RETURN;
END_IF
nCount := _Json.GetArraySize(ModulesNode);
IF nCount > Param_Config.MaxTotalConfiguredModules THEN
	ErrorMessage := CONCAT(
		CONCAT('Configuration contains more than ', TO_STRING(Param_Config.MaxTotalConfiguredModules)),
		' modules.');
	RETURN;
END_IF
_Config.ModuleCount := UDINT_TO_UINT(nCount);

FOR nModule := 1 TO _Config.ModuleCount DO
	ModuleNode := _Json.GetArrayValueByIdx(ModulesNode, UINT_TO_UDINT(nModule - 1));
	IF ModuleNode = 0 THEN
		ErrorMessage := 'Invalid module object.';
		RETURN;
	END_IF

	Node := _Json.FindMember(ModuleNode, 'enabled');
	IF Node = 0 THEN
		ErrorMessage := 'Every module requires enabled.';
		RETURN;
	END_IF
	_Config.Modules[nModule].Enabled := _Json.GetBool(Node);

	Node := _Json.FindMember(ModuleNode, 'slot');
	IF Node = 0 THEN
		ErrorMessage := 'Every module requires slot.';
		RETURN;
	END_IF
	_Config.Modules[nModule].Slot := UDINT_TO_UINT(_Json.GetUint(Node));

	Node := _Json.FindMember(ModuleNode, 'id');
	IF Node <> 0 THEN
		_Config.Modules[nModule].Id := _Json.GetUint(Node);
	END_IF
	Node := _Json.FindMember(ModuleNode, 'moduleType');
	IF Node <> 0 THEN
		_Config.Modules[nModule].ModuleType := _Json.GetString(Node);
	END_IF
	// Input mappings
	ArrayNode := _Json.FindMember(ModuleNode, 'inputMappings');
	IF ArrayNode <> 0 THEN
		nCount := _Json.GetArraySize(ArrayNode);
		IF nCount > Param_Config.MaxModuleMappings THEN
			ErrorMessage := 'Too many inputMappings.';
			RETURN;
		END_IF
		_Config.Modules[nModule].InputMappingCount := UDINT_TO_UINT(nCount);
		FOR nItem := 1 TO _Config.Modules[nModule].InputMappingCount DO
			ItemNode := _Json.GetArrayValueByIdx(ArrayNode, UINT_TO_UDINT(nItem - 1));
			Node := _Json.FindMember(ItemNode, 'source');
			IF Node <> 0 THEN _Config.Modules[nModule].InputMappings[nItem].Source := _Json.GetString(Node); END_IF
			Node := _Json.FindMember(ItemNode, 'target');
			IF Node <> 0 THEN _Config.Modules[nModule].InputMappings[nItem].Target := _Json.GetString(Node); END_IF
			Node := _Json.FindMember(ItemNode, 'sourceDataType');
			IF Node <> 0 THEN _Config.Modules[nModule].InputMappings[nItem].SourceDataType := M_ParseDataType(Value := _Json.GetString(Node)); END_IF
			Node := _Json.FindMember(ItemNode, 'targetDataType');
			IF Node <> 0 THEN _Config.Modules[nModule].InputMappings[nItem].TargetDataType := M_ParseDataType(Value := _Json.GetString(Node)); END_IF
			_Config.Modules[nModule].InputMappings[nItem].Scale := 1.0;
			TransformNode := _Json.FindMember(ItemNode, 'transform');
			IF TransformNode <> 0 THEN
				_Config.Modules[nModule].InputMappings[nItem].HasTransform := TRUE;
				Node := _Json.FindMember(TransformNode, 'scale');
				IF Node <> 0 THEN _Config.Modules[nModule].InputMappings[nItem].Scale := _Json.GetDouble(Node); END_IF
				Node := _Json.FindMember(TransformNode, 'offset');
				IF Node <> 0 THEN _Config.Modules[nModule].InputMappings[nItem].Offset := _Json.GetDouble(Node); END_IF
			END_IF
		END_FOR
	END_IF

	// Output mappings
	ArrayNode := _Json.FindMember(ModuleNode, 'outputMappings');
	IF ArrayNode <> 0 THEN
		nCount := _Json.GetArraySize(ArrayNode);
		IF nCount > Param_Config.MaxModuleMappings THEN
			ErrorMessage := 'Too many outputMappings.';
			RETURN;
		END_IF
		_Config.Modules[nModule].OutputMappingCount := UDINT_TO_UINT(nCount);
		FOR nItem := 1 TO _Config.Modules[nModule].OutputMappingCount DO
			ItemNode := _Json.GetArrayValueByIdx(ArrayNode, UINT_TO_UDINT(nItem - 1));
			Node := _Json.FindMember(ItemNode, 'source');
			IF Node <> 0 THEN _Config.Modules[nModule].OutputMappings[nItem].Source := _Json.GetString(Node); END_IF
			Node := _Json.FindMember(ItemNode, 'target');
			IF Node <> 0 THEN _Config.Modules[nModule].OutputMappings[nItem].Target := _Json.GetString(Node); END_IF
			Node := _Json.FindMember(ItemNode, 'sourceDataType');
			IF Node <> 0 THEN _Config.Modules[nModule].OutputMappings[nItem].SourceDataType := M_ParseDataType(Value := _Json.GetString(Node)); END_IF
			Node := _Json.FindMember(ItemNode, 'targetDataType');
			IF Node <> 0 THEN _Config.Modules[nModule].OutputMappings[nItem].TargetDataType := M_ParseDataType(Value := _Json.GetString(Node)); END_IF
			_Config.Modules[nModule].OutputMappings[nItem].Scale := 1.0;
			TransformNode := _Json.FindMember(ItemNode, 'transform');
			IF TransformNode <> 0 THEN
				_Config.Modules[nModule].OutputMappings[nItem].HasTransform := TRUE;
				Node := _Json.FindMember(TransformNode, 'scale');
				IF Node <> 0 THEN _Config.Modules[nModule].OutputMappings[nItem].Scale := _Json.GetDouble(Node); END_IF
				Node := _Json.FindMember(TransformNode, 'offset');
				IF Node <> 0 THEN _Config.Modules[nModule].OutputMappings[nItem].Offset := _Json.GetDouble(Node); END_IF
			END_IF
		END_FOR
	END_IF

	// Schema v4 uses a semantic name-to-source map for Module references.
	Node := _Json.FindMember(ModuleNode, 'axisReferences');
	IF Node <> 0 THEN
		ErrorMessage := 'axisReferences is not supported by schemaVersion 4; use references.';
		RETURN;
	END_IF
	Node := _Json.FindMember(ModuleNode, 'referenceBindings');
	IF Node <> 0 THEN
		ErrorMessage := 'referenceBindings is not supported by schemaVersion 4; use references.';
		RETURN;
	END_IF

	ReferencesNode := _Json.FindMember(ModuleNode, 'references');
	IF ReferencesNode <> 0 THEN
		IF NOT _Json.IsObject(ReferencesNode) THEN
			ErrorMessage := 'references must be a JSON object.';
			RETURN;
		END_IF

		nCount := 0;
		ReferenceIterator := _Json.MemberBegin(ReferencesNode);
		ReferenceIteratorEnd := _Json.MemberEnd(ReferencesNode);
		WHILE ReferenceIterator <> ReferenceIteratorEnd DO
			nCount := nCount + 1;
			IF nCount > Param_Config.MaxModuleReferences THEN
				ErrorMessage := 'Too many Module references.';
				RETURN;
			END_IF
			nItem := UDINT_TO_UINT(nCount);

			sValue := _Json.GetMemberName(ReferenceIterator);
			IF (sValue = '') OR (LEN(sValue) > 80) THEN
				ErrorMessage := 'Every Module reference requires a non-empty name of at most 80 characters.';
				RETURN;
			END_IF
			IF nItem > 1 THEN
				FOR nOther := 1 TO nItem - 1 DO
					IF _Config.Modules[nModule].References[nOther].Name = sValue THEN
						ErrorMessage := CONCAT('Duplicate Module reference name: ', sValue);
						RETURN;
					END_IF
				END_FOR
			END_IF

			ItemNode := _Json.GetMemberValue(ReferenceIterator);
			IF (ItemNode = 0) OR NOT _Json.IsString(ItemNode) THEN
				ErrorMessage := CONCAT('Module reference source must be a string: ', sValue);
				RETURN;
			END_IF
			_Config.Modules[nModule].References[nItem].Name := sValue;
			_Config.Modules[nModule].References[nItem].Source := _Json.GetString(ItemNode);
			IF _Config.Modules[nModule].References[nItem].Source = '' THEN
				ErrorMessage := CONCAT('Module reference source must not be empty: ', sValue);
				RETURN;
			END_IF

			ReferenceIterator := _Json.NextMember(ReferenceIterator);
		END_WHILE
		_Config.Modules[nModule].ReferenceCount := UDINT_TO_UINT(nCount);
	END_IF

	// Variable list
	ArrayNode := _Json.FindMember(ModuleNode, 'variableList');
	IF ArrayNode <> 0 THEN
		nCount := _Json.GetArraySize(ArrayNode);
		IF nCount > Param_Config.MaxModuleVariable THEN
			ErrorMessage := 'Too many variableList entries.';
			RETURN;
		END_IF
		_Config.Modules[nModule].VariableCount := UDINT_TO_UINT(nCount);
		FOR nItem := 1 TO _Config.Modules[nModule].VariableCount DO
			ItemNode := _Json.GetArrayValueByIdx(ArrayNode, UINT_TO_UDINT(nItem - 1));
			Node := _Json.FindMember(ItemNode, 'source');
			IF Node <> 0 THEN _Config.Modules[nModule].VariableList[nItem].Source := _Json.GetString(Node); END_IF
			Node := _Json.FindMember(ItemNode, 'id');
			IF Node <> 0 THEN _Config.Modules[nModule].VariableList[nItem].Id := _Json.GetUint(Node); END_IF
			Node := _Json.FindMember(ItemNode, 'name');
			IF Node <> 0 THEN _Config.Modules[nModule].VariableList[nItem].Name := _Json.GetString(Node); END_IF
			Node := _Json.FindMember(ItemNode, 'unit');
			IF Node <> 0 THEN _Config.Modules[nModule].VariableList[nItem].Unit := _Json.GetString(Node); END_IF
			Node := _Json.FindMember(ItemNode, 'dataType');
			IF Node <> 0 THEN _Config.Modules[nModule].VariableList[nItem].DataType := M_ParseDataType(Value := _Json.GetString(Node)); END_IF
		END_FOR
	END_IF

	// Alarm list; condition is an object to avoid parsing a mini expression language.
	ArrayNode := _Json.FindMember(ModuleNode, 'alarmList');
	IF ArrayNode <> 0 THEN
		nCount := _Json.GetArraySize(ArrayNode);
		IF nCount > Param_Config.MaxConfiguredAlarmsPerModule THEN
			ErrorMessage := 'Too many alarmList entries.';
			RETURN;
		END_IF
		_Config.Modules[nModule].AlarmCount := UDINT_TO_UINT(nCount);
		FOR nItem := 1 TO _Config.Modules[nModule].AlarmCount DO
			ItemNode := _Json.GetArrayValueByIdx(ArrayNode, UINT_TO_UDINT(nItem - 1));
			Node := _Json.FindMember(ItemNode, 'source');
			IF Node <> 0 THEN _Config.Modules[nModule].AlarmList[nItem].Source := _Json.GetString(Node); END_IF
			Node := _Json.FindMember(ItemNode, 'dataType');
			IF Node <> 0 THEN _Config.Modules[nModule].AlarmList[nItem].DataType := M_ParseDataType(Value := _Json.GetString(Node)); END_IF
			ConditionNode := _Json.FindMember(ItemNode, 'condition');
			IF ConditionNode = 0 THEN
				ErrorMessage := 'Every alarm requires a condition object.';
				RETURN;
			END_IF
			Node := _Json.FindMember(ConditionNode, 'operator');
			IF Node <> 0 THEN _Config.Modules[nModule].AlarmList[nItem].Operator := M_ParseOperator(Value := _Json.GetString(Node)); END_IF
			Node := _Json.FindMember(ConditionNode, 'value');
			IF Node <> 0 THEN _Config.Modules[nModule].AlarmList[nItem].Threshold := _Json.GetDouble(Node); END_IF
			Node := _Json.FindMember(ConditionNode, 'tolerance');
			IF Node <> 0 THEN _Config.Modules[nModule].AlarmList[nItem].Tolerance := _Json.GetDouble(Node); END_IF
			Node := _Json.FindMember(ItemNode, 'mainErrorId');
			IF Node <> 0 THEN _Config.Modules[nModule].AlarmList[nItem].MainErrorId := _Json.GetUint(Node); END_IF
			Node := _Json.FindMember(ItemNode, 'sourceErrorId');
			IF Node <> 0 THEN _Config.Modules[nModule].AlarmList[nItem].SourceErrorId := _Json.GetUint(Node); END_IF
			Node := _Json.FindMember(ItemNode, 'message');
			IF Node <> 0 THEN _Config.Modules[nModule].AlarmList[nItem].Message := _Json.GetString(Node); END_IF
			Node := _Json.FindMember(ItemNode, 'severity');
			IF Node <> 0 THEN
				sValue := _Json.GetString(Node);
				_Config.Modules[nModule].AlarmList[nItem].Severity := M_ParseSeverity(Value := sValue);
			ELSE
				_Config.Modules[nModule].AlarmList[nItem].Severity := E_Severity.Alarm;
			END_IF
		END_FOR
	END_IF
END_FOR

IF NOT M_ValidateParsedConfiguration() THEN
	RETURN;
END_IF
M_ParseDocument := TRUE;
END_METHOD

METHOD PRIVATE M_ParseOperator : E_AlarmOperator
VAR_INPUT
	Value : STRING(255);
END_VAR
IF Value = 'gt' THEN M_ParseOperator := E_AlarmOperator.GreaterThan;
ELSIF Value = 'lt' THEN M_ParseOperator := E_AlarmOperator.LessThan;
ELSIF Value = 'eq' THEN M_ParseOperator := E_AlarmOperator.Equal;
ELSIF Value = 'ge' THEN M_ParseOperator := E_AlarmOperator.GreaterOrEqual;
ELSIF Value = 'le' THEN M_ParseOperator := E_AlarmOperator.LessOrEqual;
ELSE M_ParseOperator := E_AlarmOperator.Invalid;
END_IF
END_METHOD

METHOD PRIVATE M_ParseSeverity : E_Severity
VAR_INPUT
	Value : STRING(255);
END_VAR
IF Value = TO_STRING(E_Severity.Warning) THEN M_ParseSeverity := E_Severity.Warning;
ELSE M_ParseSeverity := E_Severity.Alarm;
END_IF
END_METHOD

METHOD PRIVATE M_ValidateParsedConfiguration : BOOL
VAR
	nModule : UINT;
	nItem : UINT;
	nOther : UINT;
END_VAR
M_ValidateParsedConfiguration := FALSE;
FOR nModule := 1 TO _Config.ModuleCount DO
	IF NOT _Config.Modules[nModule].Enabled THEN
		CONTINUE;
	END_IF
	FOR nItem := 1 TO _Config.Modules[nModule].InputMappingCount DO
		IF (_Config.Modules[nModule].InputMappings[nItem].Source = '')
			OR (_Config.Modules[nModule].InputMappings[nItem].Target = '')
			OR (_Config.Modules[nModule].InputMappings[nItem].SourceDataType = E_ConfigDataType.Unknown)
			OR (_Config.Modules[nModule].InputMappings[nItem].TargetDataType = E_ConfigDataType.Unknown) THEN
			ErrorMessage := 'Invalid input mapping: source, target and both data types are required.';
			RETURN;
		END_IF
	END_FOR
	FOR nItem := 1 TO _Config.Modules[nModule].OutputMappingCount DO
		IF (_Config.Modules[nModule].OutputMappings[nItem].Source = '')
			OR (_Config.Modules[nModule].OutputMappings[nItem].Target = '')
			OR (_Config.Modules[nModule].OutputMappings[nItem].SourceDataType = E_ConfigDataType.Unknown)
			OR (_Config.Modules[nModule].OutputMappings[nItem].TargetDataType = E_ConfigDataType.Unknown) THEN
			ErrorMessage := 'Invalid output mapping: source, target and both data types are required.';
			RETURN;
		END_IF
	END_FOR
	FOR nItem := 1 TO _Config.Modules[nModule].ReferenceCount DO
		IF (_Config.Modules[nModule].References[nItem].Name = '')
			OR (_Config.Modules[nModule].References[nItem].Source = '') THEN
			ErrorMessage := 'Invalid Module reference: name and source are required.';
			RETURN;
		END_IF
	END_FOR
	FOR nItem := 1 TO _Config.Modules[nModule].VariableCount DO
		IF (_Config.Modules[nModule].VariableList[nItem].Source = '')
			OR (_Config.Modules[nModule].VariableList[nItem].Id = 0)
			OR (_Config.Modules[nModule].VariableList[nItem].DataType = E_ConfigDataType.Unknown) THEN
			ErrorMessage := 'Invalid variableList entry.';
			RETURN;
		END_IF
	END_FOR
	FOR nItem := 1 TO _Config.Modules[nModule].AlarmCount DO
		IF (_Config.Modules[nModule].AlarmList[nItem].Source = '')
			OR (_Config.Modules[nModule].AlarmList[nItem].DataType = E_ConfigDataType.Unknown)
			OR (_Config.Modules[nModule].AlarmList[nItem].Operator = E_AlarmOperator.Invalid)
			OR (_Config.Modules[nModule].AlarmList[nItem].MainErrorId = 0) THEN
			ErrorMessage := 'Invalid alarmList entry.';
			RETURN;
		END_IF
		FOR nOther := nItem + 1 TO _Config.Modules[nModule].AlarmCount DO
			IF _Config.Modules[nModule].AlarmList[nItem].MainErrorId
				= _Config.Modules[nModule].AlarmList[nOther].MainErrorId THEN
				ErrorMessage := 'Duplicate configured alarm mainErrorId in module.';
				RETURN;
			END_IF
		END_FOR
	END_FOR
END_FOR
M_ValidateParsedConfiguration := TRUE;
END_METHOD

END_FUNCTION_BLOCK

// ---- Configuration/POUs/FB_ApplicationConfigRoot.TcPOU
FUNCTION_BLOCK ABSTRACT FB_ApplicationConfigRoot
VAR
	_LinkVariableManager : FB_LinkVariableManager;
	_ReferenceManager : FB_ReferenceManager;
	_ModuleTypeRegistry : FB_ModuleTypeRegistry;
	_ModuleConfigurationManager : FB_ModuleConfigurationManager;
	_UtcClock : FB_UtcClock;
	_SystemContext : ST_SystemContext;
	_bRegistrationAttempted : BOOL;
	_bRegistered : BOOL;
	_bError : BOOL;
	_hrErrorCode : HRESULT;
	_sErrorMessage : STRING(255);
END_VAR

PROPERTY PUBLIC FINAL Busy : BOOL
GET
Busy := _bRegistered AND NOT _bError AND _ModuleConfigurationManager.Busy;
END_GET
END_PROPERTY

PROPERTY PUBLIC FINAL Error : BOOL
GET
Error := _bError;
END_GET
END_PROPERTY

PROPERTY PUBLIC FINAL ErrorCode : HRESULT
GET
ErrorCode := _hrErrorCode;
END_GET
END_PROPERTY

PROPERTY PUBLIC FINAL ErrorMessage : STRING(255)
GET
ErrorMessage := _sErrorMessage;
END_GET
END_PROPERTY

METHOD PROTECTED H_RegisterBaseUnits
END_METHOD

METHOD PROTECTED H_RegisterIo
END_METHOD

METHOD PROTECTED H_RegisterModuleTypes
END_METHOD

METHOD PROTECTED H_RunModules
VAR_INPUT
	VariableNodeReader : I_VariableNodeReader;
END_VAR
VAR_IN_OUT CONSTANT
	SystemContext : ST_SystemContext;
END_VAR
END_METHOD

METHOD PUBLIC FINAL Run
M_PollConfiguration();

_UtcClock(UtcDateTime => _SystemContext.UtcDateTime);
_SystemContext.ModuleHeartbeatTimeout := Param_Config.ModuleHeartbeat_Timeout;

IF Ready THEN
	_LinkVariableManager.M_CyclicInput();
	H_RunModules(
		SystemContext := _SystemContext,
		VariableNodeReader := _LinkVariableManager);
	_LinkVariableManager.M_CyclicOutput();
END_IF
END_METHOD

METHOD PRIVATE M_PollConfiguration
VAR
	bRegistrationSessionStarted : BOOL;
	bRegistrationSealed : BOOL;
END_VAR
IF NOT _bRegistrationAttempted THEN
	_bRegistrationAttempted := TRUE;

	// The base class owns the Infrastructure registration session.
	bRegistrationSessionStarted := _LinkVariableManager.M_BeginInfrastructureRegistration();
	IF NOT bRegistrationSessionStarted THEN
		M_SetError(
			Message := _LinkVariableManager.ErrorMessage,
			ErrorCode := 0);
	ELSE
		H_RegisterIo();

		// Always seal an opened session. On a registration error this also rolls
		// back every Infrastructure node declared during this attempt.
		bRegistrationSealed := _LinkVariableManager.M_SealInfrastructureRegistration();
		IF NOT bRegistrationSealed THEN
			M_SetError(
				Message := _LinkVariableManager.ErrorMessage,
				ErrorCode := 0);
		END_IF
	END_IF

	IF NOT _bError THEN
		H_RegisterBaseUnits();
	END_IF
	IF NOT _bError THEN
		H_RegisterModuleTypes();
	END_IF

	_bRegistered := NOT _bError;
END_IF

IF NOT _bRegistered OR _bError THEN
	RETURN;
END_IF

_ModuleConfigurationManager(
	Execute := TRUE,
	FilePath := Param_Config.ModuleConfigFilePath,
	LinkVariableManager := _LinkVariableManager,
	ReferenceManager := _ReferenceManager,
	ModuleTypeRegistry := _ModuleTypeRegistry);

IF _ModuleConfigurationManager.Error THEN
	M_SetError(
		Message := _ModuleConfigurationManager.ErrorMessage,
		ErrorCode := _ModuleConfigurationManager.ErrorCode);
END_IF
END_METHOD

METHOD PROTECTED FINAL M_RegisterBaseUnit : BOOL
VAR_INPUT
	BaseUnit : I_BaseUnit;
END_VAR
M_RegisterBaseUnit := FALSE;
IF _bError THEN
	RETURN;
END_IF

M_RegisterBaseUnit := _ReferenceManager.M_RegisterReference(BaseUnit := BaseUnit);
IF NOT M_RegisterBaseUnit THEN
	M_SetError(
		Message := _ReferenceManager.ErrorMessage,
		ErrorCode := 0);
END_IF
END_METHOD

METHOD PROTECTED FINAL M_RegisterIoNode : BOOL
VAR_INPUT
	Variable : ANY;
	Access : E_VariableAccess;
END_VAR
M_RegisterIoNode := FALSE;
IF _bError THEN
	RETURN;
END_IF

M_RegisterIoNode := _LinkVariableManager.M_RegisterInfrastructureNode(
	Variable := Variable,
	Access := Access);
IF NOT M_RegisterIoNode THEN
	M_SetError(
		Message := _LinkVariableManager.ErrorMessage,
		ErrorCode := 0);
END_IF
END_METHOD

METHOD PROTECTED FINAL M_RegisterModuleType : BOOL
VAR_INPUT
	ModuleTypeName : T_ModuleTypeName;
	Adapter : I_ModuleConfigurationAdapter;
END_VAR
M_RegisterModuleType := FALSE;
IF _bError THEN
	RETURN;
END_IF

M_RegisterModuleType := _ModuleTypeRegistry.M_Register(
	ModuleTypeName := ModuleTypeName,
	Adapter := Adapter);
IF NOT M_RegisterModuleType THEN
	M_SetError(
		Message := _ModuleTypeRegistry.ErrorMessage,
		ErrorCode := 0);
END_IF
END_METHOD

METHOD PRIVATE M_SetError
VAR_INPUT
	Message : STRING(255);
	ErrorCode : HRESULT;
END_VAR
IF NOT _bError THEN
	_bError := TRUE;
	_hrErrorCode := ErrorCode;
	IF Message = '' THEN
		_sErrorMessage := 'Application configuration initialization failed.';
	ELSE
		_sErrorMessage := Message;
	END_IF
END_IF
END_METHOD

PROPERTY PUBLIC FINAL Ready : BOOL
GET
Ready := _bRegistered AND NOT _bError AND _ModuleConfigurationManager.Ready;
END_GET
END_PROPERTY

END_FUNCTION_BLOCK

// ---- POUs/00_BaseUnit/FB_Axis_BaseUnit.TcPOU
FUNCTION_BLOCK FB_Axis_BaseUnit EXTENDS FB_BaseUnit IMPLEMENTS I_Axis_BaseUnit
VAR_INPUT
END_VAR
VAR_OUTPUT
END_VAR

VAR
	_Axis		: AXIS_REF;
	_MCMoveAbs	: MC_MoveAbsolute;
	_MCReset	: MC_Reset;
	_MCStop		: MC_Stop;
	_MCMoveVel	: MC_MoveVelocity;
	_MCMoveVel_2 : MC_MoveVelocity;
	_VelSwitchTrig : F_TRIG;
	_bVelSwitch : BOOL;
	_MCPower	: MC_Power;
	_MCJog		: MC_Jog;
	_MCHalt		: MC_Halt;
END_VAR

M_CyclicUpdate();

PROPERTY PUBLIC AxisActualPosition : LREAL
GET
// Expose motion feedback without exposing AXIS_REF to Services.
AxisActualPosition := _Axis.NcToPlc.ActPos;
END_GET
END_PROPERTY

PROPERTY PUBLIC AxisActualVelocity : LREAL
GET
// Expose motion feedback without exposing AXIS_REF to Services.
AxisActualVelocity := _Axis.NcToPlc.ActVelo;
END_GET
END_PROPERTY

PROPERTY PUBLIC AxisHasJob : BOOL
GET
// Expose motion feedback without exposing AXIS_REF to Services.
AxisHasJob := _Axis.Status.HasJob;
END_GET
END_PROPERTY

PROPERTY PUBLIC AxisIsDisabled : BOOL
GET
// Treat an invalid Axis reference as unavailable to callers.
AxisIsDisabled := _Axis.Status.Disabled;
END_GET
END_PROPERTY

METHOD M_CyclicUpdate
VAR_INPUT
END_VAR
_MCPower(Axis:= _Axis,
			Enable:= TRUE,
			Enable_Positive:= TRUE,
			Enable_Negative:= TRUE,
			Override:= 100);
			
_MCReset(Axis:= _Axis);
_MCStop(Axis:= _Axis);
_MCMoveAbs(Axis:= _Axis);
_MCMoveVel(Axis:= _Axis);
_MCMoveVel_2(Axis:= _Axis);
_MCJog(Axis:= _Axis);
_MCHalt(Axis:= _Axis);

_Axis.ReadStatus();
END_METHOD

METHOD M_Halt : BOOL
VAR_INPUT
	OwnerId : T_ResourceOwnerId;
	Execute : BOOL;
	Deceleration : LREAL;
END_VAR
VAR_OUTPUT
	Done : BOOL;
	Error : BOOL;
END_VAR
M_Halt := FALSE;
Done := FALSE;
Error := FALSE;
IF NOT M_IsResourceOwner(OwnerId := OwnerId) THEN
	RETURN;
END_IF

_MCHalt.Execute := Execute;
_MCHalt.Deceleration := Deceleration;

Done := _MCHalt.Done;
Error := _MCHalt.Error;
M_Halt := TRUE;
END_METHOD

METHOD M_Jog : BOOL
VAR_INPUT
	OwnerId : T_ResourceOwnerId;
	JogForward : BOOL;
	JogBackwards : BOOL;
	Mode : E_JogMode;
	Position : LREAL;
	Velocity : LREAL;
	Acceleration : LREAL;
	Deceleration : LREAL;
END_VAR

VAR_OUTPUT
	Done : BOOL;
	Error : BOOL;
	ErrorId : UDINT;
END_VAR
// Ignore commands from Services that do not own this BaseUnit.
M_Jog := FALSE;
Done := FALSE;
Error := FALSE;
ErrorId := 0;
IF NOT M_IsResourceOwner(OwnerId := OwnerId) THEN
	RETURN;
END_IF

_MCJog.JogForward := JogForward;
_MCJog.JogBackwards := JogBackwards;
_MCJog.Mode := Mode;
_MCJog.Position := Position;
_MCJog.Velocity := Velocity;
_MCJog.Acceleration := Acceleration;
_MCJog.Deceleration := Deceleration;

Done := _MCJog.Done;
Error := _MCJog.Error;
ErrorId := _MCJog.ErrorId;
M_Jog := TRUE;
END_METHOD

METHOD M_MoveAbs : BOOL
VAR_INPUT
	OwnerId : T_ResourceOwnerId;
	Execute : BOOL;
	Position : LREAL;
	Velocity : LREAL;
	Acceleration : LREAL;
	Deceleration : LREAL;
END_VAR

VAR_OUTPUT
	Done : BOOL;
	Error : BOOL;
	ErrorId : UDINT;
END_VAR
// Ignore commands from Services that do not own this BaseUnit.
M_MoveAbs := FALSE;
Done := FALSE;
Error := FALSE;
ErrorId := 0;
IF NOT M_IsResourceOwner(OwnerId := OwnerId) THEN
	RETURN;
END_IF

_MCMoveAbs.Execute := Execute;
_MCMoveAbs.Position := Position;
_MCMoveAbs.Velocity := Velocity;
_MCMoveAbs.Acceleration := Acceleration;
_MCMoveAbs.Deceleration := Deceleration;

Done := _MCMoveAbs.Done;
Error := _MCMoveAbs.Error;
ErrorId := _MCMoveAbs.ErrorId;
M_MoveAbs := TRUE;
END_METHOD

METHOD M_MoveVel : BOOL
VAR_INPUT
	OwnerId : T_ResourceOwnerId;
	Execute : BOOL;
	Direction : MC_Direction;
	Velocity : LREAL;
	Acceleration : LREAL;
	Deceleration : LREAL;
END_VAR

VAR_OUTPUT
	InVelocity : BOOL;
	Error : BOOL;
END_VAR
// Ignore commands from Services that do not own this BaseUnit.
M_MoveVel := FALSE;
InVelocity := FALSE;
Error := FALSE;
IF NOT M_IsResourceOwner(OwnerId := OwnerId) THEN
	RETURN;
END_IF

// Clear input
IF Execute = FALSE THEN
	_MCMoveVel.Execute := FALSE;
	_MCMoveVel_2.Execute := FALSE;
END_IF

// Switch MoveVelocity when falling trig
_VelSwitchTrig(CLK:= Execute, Q=> );
IF _VelSwitchTrig.Q THEN
	_bVelSwitch := NOT _bVelSwitch;
END_IF

IF _bVelSwitch THEN
	_MCMoveVel.Execute := Execute;
	_MCMoveVel.Direction := Direction;
	_MCMoveVel.Velocity := Velocity;
	_MCMoveVel.Acceleration := Acceleration;
	_MCMoveVel.Deceleration := Deceleration;
	InVelocity := _MCMoveVel.InVelocity;
	Error := _MCMoveVel.Error;
ELSE
	_MCMoveVel_2.Execute := Execute;
	_MCMoveVel_2.Direction := Direction;
	_MCMoveVel_2.Velocity := Velocity;
	_MCMoveVel_2.Acceleration := Acceleration;
	_MCMoveVel_2.Deceleration := Deceleration;
	InVelocity := _MCMoveVel_2.InVelocity;
	Error := _MCMoveVel_2.Error;
	
END_IF

M_MoveVel := TRUE;
END_METHOD

METHOD M_Reset : BOOL
VAR_INPUT
	OwnerId : T_ResourceOwnerId;
	Execute : BOOL;
END_VAR

VAR_OUTPUT
	Done : BOOL;
	Error : BOOL;
	ErrorId : UDINT;
END_VAR
// Ignore commands from Services that do not own this BaseUnit.
M_Reset := FALSE;
Done := FALSE;
Error := FALSE;
ErrorId := 0;
IF NOT M_IsResourceOwner(OwnerId := OwnerId) THEN
	RETURN;
END_IF

_MCReset.Execute := Execute;

Done := _MCReset.Done;
Error := _MCReset.Error;
ErrorId := _MCReset.ErrorId;
M_Reset := TRUE;
END_METHOD

METHOD M_Stop : BOOL
VAR_INPUT
	OwnerId : T_ResourceOwnerId;
	Execute : BOOL;
	Deceleration : LREAL;
END_VAR

VAR_OUTPUT
	Done : BOOL;
	Error : BOOL;
	ErrorId : UDINT;
END_VAR
M_Stop := FALSE;
Done := FALSE;
Error := FALSE;
ErrorId := 0;
IF NOT M_IsResourceOwner(OwnerId := OwnerId) THEN
	RETURN;
END_IF

_MCStop.Execute := Execute;
_MCStop.Deceleration := Deceleration;

Done := _MCStop.Done;
Error := _MCStop.Error;
ErrorId := _MCStop.ErrorId;
M_Stop := TRUE;
END_METHOD

END_FUNCTION_BLOCK

// ---- POUs/10_Module/FB_ModuleAlarmManager.TcPOU
FUNCTION_BLOCK FB_ModuleAlarmManager
VAR_OUTPUT
	AckResponseId : UDINT;
	AckAccepted : BOOL;
	AckError : E_AlarmAckError;
	ConfiguredLatchedCount : UINT;
	ServiceLatchedCount : UINT;
	Overflow : BOOL;
	HookLatchedCount : UINT;
	DuplicateId : UDINT;
END_VAR
VAR
	_ConfiguredStates : ARRAY[1..Param_Config.MaxConfiguredAlarmsPerModule] OF ST_AlarmLifecycleState;
	_ServiceStates : ARRAY[1..Param_Config.MaxServiceAlarmsPerModule] OF ST_AlarmLifecycleState;
	_HookStates : ARRAY[1..Param_Config.MaxHookAlarmsPerModule] OF ST_AlarmLifecycleState;
	_AckRequestOneShot : R_TRIG;
	_LastAckRequestId : UDINT;
	_ModuleId : UDINT;
	_ConfigurationRevision : UDINT;
END_VAR

METHOD PRIVATE M_AcknowledgeState
VAR_IN_OUT
	State : ST_AlarmLifecycleState;
END_VAR
State.Alarm.Acknowledged := TRUE;
IF NOT State.Alarm.Active THEN
	MEMSET(ADR(State), 0, SIZEOF(State));
END_IF
END_METHOD

METHOD PUBLIC M_BeginCycle
VAR_INPUT
	ModuleId : UDINT;
	ConfigurationRevision : UDINT;
END_VAR
VAR
	nIndex : UINT;
END_VAR
IF ModuleId <> _ModuleId THEN
	MEMSET(ADR(_ConfiguredStates), 0, SIZEOF(_ConfiguredStates));
	MEMSET(ADR(_ServiceStates), 0, SIZEOF(_ServiceStates));
	MEMSET(ADR(_HookStates), 0, SIZEOF(_HookStates));
	M_ResetAcknowledgement();
	_ModuleId := ModuleId;
	_ConfigurationRevision := ConfigurationRevision;

ELSIF ConfigurationRevision <> _ConfigurationRevision THEN
	// Reset JSON lifecycles; the Module suppresses only Hook identities taken over by JSON.
	MEMSET(ADR(_ConfiguredStates), 0, SIZEOF(_ConfiguredStates));
	_ConfigurationRevision := ConfigurationRevision;
END_IF

Overflow := FALSE;
DuplicateId := 0;
FOR nIndex := 1 TO Param_Config.MaxServiceAlarmsPerModule DO
	_ServiceStates[nIndex].SeenThisCycle := FALSE;
END_FOR
FOR nIndex := 1 TO Param_Config.MaxHookAlarmsPerModule DO
	_HookStates[nIndex].SeenThisCycle := FALSE;
END_FOR
END_METHOD

METHOD PUBLIC M_EndCycle
VAR
	nIndex : UINT;
END_VAR
FOR nIndex := 1 TO Param_Config.MaxServiceAlarmsPerModule DO
	IF NOT _ServiceStates[nIndex].Latched THEN
		CONTINUE;
	END_IF

	IF NOT _ServiceStates[nIndex].SeenThisCycle THEN
		_ServiceStates[nIndex].Alarm.Active := FALSE;
	END_IF

	IF NOT _ServiceStates[nIndex].Alarm.Active
		AND _ServiceStates[nIndex].Alarm.Acknowledged THEN
		MEMSET(ADR(_ServiceStates[nIndex]), 0, SIZEOF(_ServiceStates[nIndex]));
	END_IF
END_FOR

FOR nIndex := 1 TO Param_Config.MaxHookAlarmsPerModule DO
	IF NOT _HookStates[nIndex].Latched THEN
		CONTINUE;
	END_IF

	IF NOT _HookStates[nIndex].SeenThisCycle THEN
		_HookStates[nIndex].Alarm.Active := FALSE;
	END_IF

	IF NOT _HookStates[nIndex].Alarm.Active
		AND _HookStates[nIndex].Alarm.Acknowledged THEN
		MEMSET(ADR(_HookStates[nIndex]), 0, SIZEOF(_HookStates[nIndex]));
	END_IF
END_FOR
END_METHOD

METHOD PRIVATE M_LatchState
VAR_INPUT
	ServiceId : UDINT;
	DateTime : STRING(20);
END_VAR
VAR_IN_OUT
	State : ST_AlarmLifecycleState;
END_VAR
VAR_IN_OUT CONSTANT
	Snapshot : ST_ExtAlarm;
END_VAR
MEMSET(ADR(State), 0, SIZEOF(State));
State.Latched := TRUE;
State.Alarm := Snapshot;
State.Alarm.ModuleId := _ModuleId;
State.Alarm.ServiceId := ServiceId;
State.Alarm.DateTime := DateTime;
State.Alarm.Active := TRUE;
State.Alarm.Acknowledged := FALSE;
State.Alarm.OccurrenceCount := 1;
END_METHOD

METHOD PUBLIC M_ObserveServiceAlarm : BOOL
VAR_IN_OUT CONSTANT
	Alarm : ST_ExtAlarm;
END_VAR
VAR
	nIndex : UINT;
	nFirstEmpty : UINT;
END_VAR
M_ObserveServiceAlarm := FALSE;
nFirstEmpty := 0;

IF (Alarm.ServiceId = 0) OR (Alarm.MainErrorId = 0) THEN
	RETURN;
END_IF

FOR nIndex := 1 TO Param_Config.MaxServiceAlarmsPerModule DO

	// If slot has been used
	IF _ServiceStates[nIndex].Latched THEN

		// If alarm has already in latched queue
		IF (_ServiceStates[nIndex].Alarm.ServiceId = Alarm.ServiceId)
			AND (_ServiceStates[nIndex].Alarm.MainErrorId = Alarm.MainErrorId) THEN
			_ServiceStates[nIndex].SeenThisCycle := TRUE;

